LIN {X 0,Y 304.363,Z 602.903,A -85,B 0,C 180,E1 -16113.309,E2 -16113.309} C_VEL
LIN {X 0,Y 304.825,Z 598.921,A -85,B 0,C 180,E1 -16115.292,E2 -16115.292} C_VEL
LIN {X 0,Y 305.684,Z 593.946,A -85,B 0,C 180,E1 -16117.265,E2 -16117.265} C_VEL
LIN {X 0,Y 306.926,Z 586.616,A -85,B 0,C 180,E1 -16119.625,E2 -16119.625} C_VEL
LIN {X 0,Y 308.147,Z 578.097,A -85,B 0,C 180,E1 -16121.845,E2 -16121.845} C_VEL
LIN {X 0,Y 309.957,Z 568.895,A -85,B 0,C 180,E1 -16123.773,E2 -16123.773} C_VEL
LIN {X 0,Y 311.67,Z 558.74,A -85,B 0,C 180,E1 -16125.532,E2 -16125.532} C_VEL
LIN {X 0,Y 313.434,Z 547.553,A -85,B 0,C 180,E1 -16127.115,E2 -16127.115} C_VEL
LIN {X 0,Y 314.915,Z 536.756,A -85,B 0,C 180,E1 -16128.375,E2 -16128.375} C_VEL
LIN {X 0,Y 316.351,Z 525.204,A -85,B 0,C 180,E1 -16129.465,E2 -16129.465} C_VEL
LIN {X 0,Y 317.646,Z 512.743,A -85,B 0,C 180,E1 -16130.394,E2 -16130.394} C_VEL
LIN {X 0,Y 318.767,Z 498.862,A -85,B 0,C 180,E1 -16131.163,E2 -16131.163} C_VEL
LIN {X 0,Y 319.468,Z 485.64,A -85,B 0,C 180,E1 -16131.665,E2 -16131.665} C_VEL
LIN {X 0,Y 322.236,Z 387.309,A -85,B 0,C 180,E1 -16133.852,E2 -16133.852} C_VEL
LIN {X 0,Y 314.712,Z 368.239,A -85,B 0,C 180,E1 -16135.033,E2 -16135.033} C_VEL
LIN {X 0,Y 307.818,Z 353.094,A -85,B 0,C 180,E1 -16136.117,E2 -16136.117} C_VEL
LIN {X 0,Y 306.342,Z 349.731,A -85,B 0,C 180,E1 -16136.399,E2 -16136.399} C_VEL
LIN {X 0,Y 305.459,Z 346.064,A -85,B 0,C 180,E1 -16137.676,E2 -16137.676} C_VEL
LIN {X 0,Y 305.437,Z 346.065,A -85,B 0,C 180,E1 -16141.953,E2 -16141.953} C_VEL
LIN {X 0,Y 305.423,Z 346.063,A -85,B 0,C 180,E1 -16142.702,E2 -16142.702} C_VEL
LIN {X 0,Y 304.77,Z 346.147,A -85,B 0,C 180,E1 -16143.803,E2 -16143.803} C_VEL
LIN {X 0,Y 301.908,Z 346.503,A -85,B 0,C 180,E1 -16145.596,E2 -16145.596} C_VEL
LIN {X 0,Y 299.479,Z 346.804,A -85,B 0,C 180,E1 -16147.05,E2 -16147.05} C_VEL
LIN {X 0,Y 298.449,Z 346.935,A -85,B 0,C 180,E1 -16148.177,E2 -16148.177} C_VEL
LIN {X 0,Y 298.372,Z 346.94,A -85,B 0,C 180,E1 -16148.559,E2 -16148.559} C_VEL
LIN {X 0,Y 298.349,Z 346.944,A -85,B 0,C 180,E1 -16151.268,E2 -16151.268} C_VEL
LIN {X 0,Y 298.357,Z 346.94,A -85,B 0,C 180,E1 -16155.035,E2 -16155.035} C_VEL
LIN {X 0,Y 298.35,Z 346.941,A -85,B 0,C 180,E1 -16158.921,E2 -16158.921} C_VEL
LIN {X 0,Y 298.429,Z 346.93,A -85,B 0,C 180,E1 -16163.197,E2 -16163.197} C_VEL
LIN {X 0,Y 298.395,Z 346.929,A -85,B 0,C 180,E1 -16167.199,E2 -16167.199} C_VEL
LIN {X 0,Y 298.366,Z 346.942,A -85,B 0,C 180,E1 -16170.638,E2 -16170.638} C_VEL
LIN {X 0,Y 298.423,Z 346.937,A -85,B 0,C 180,E1 -16174.918,E2 -16174.918} C_VEL
LIN {X 0,Y 298.401,Z 346.924,A -85,B 0,C 180,E1 -16177.862,E2 -16177.862} C_VEL
LIN {X 0,Y 298.462,Z 346.907,A -85,B 0,C 180,E1 -16180.751,E2 -16180.751} C_VEL
LIN {X 0,Y 298.513,Z 346.923,A -85,B 0,C 180,E1 -16184.99,E2 -16184.99} C_VEL
LIN {X 0,Y 298.585,Z 346.881,A -85,B 0,C 180,E1 -16189.146,E2 -16189.146} C_VEL
LIN {X 0,Y 298.7,Z 346.893,A -85,B 0,C 180,E1 -16191.884,E2 -16191.884} C_VEL
LIN {X 0,Y 298.637,Z 346.908,A -85,B 0,C 180,E1 -16194.598,E2 -16194.598} C_VEL
LIN {X 0,Y 298.909,Z 346.876,A -85,B 0,C 180,E1 -16198.652,E2 -16198.652} C_VEL
LIN {X 0,Y 298.916,Z 346.867,A -85,B 0,C 180,E1 -16201.347,E2 -16201.347} C_VEL
LIN {X 0,Y 298.738,Z 346.896,A -85,B 0,C 180,E1 -16206.755,E2 -16206.755} C_VEL
LIN {X 0,Y 298.628,Z 346.909,A -85,B 0,C 180,E1 -16209.482,E2 -16209.482} C_VEL
LIN {X 0,Y 298.555,Z 346.918,A -85,B 0,C 180,E1 -16213.615,E2 -16213.615} C_VEL
LIN {X 0,Y 298.551,Z 346.921,A -85,B 0,C 180,E1 -16216.408,E2 -16216.408} C_VEL
LIN {X 0,Y 298.513,Z 346.925,A -85,B 0,C 180,E1 -16219.654,E2 -16219.654} C_VEL
LIN {X 0,Y 298.428,Z 346.937,A -85,B 0,C 180,E1 -16223.6,E2 -16223.6} C_VEL
LIN {X 0,Y 298.455,Z 346.933,A -85,B 0,C 180,E1 -16226.577,E2 -16226.577} C_VEL
LIN {X 0,Y 298.404,Z 346.938,A -85,B 0,C 180,E1 -16229.643,E2 -16229.643} C_VEL
LIN {X 0,Y 298.394,Z 346.939,A -85,B 0,C 180,E1 -16232.8,E2 -16232.8} C_VEL
LIN {X 0,Y 298.466,Z 346.934,A -85,B 0,C 180,E1 -16236.812,E2 -16236.812} C_VEL
LIN {X 0,Y 298.388,Z 346.944,A -85,B 0,C 180,E1 -16241.087,E2 -16241.087} C_VEL
LIN {X 0,Y 298.399,Z 346.943,A -85,B 0,C 180,E1 -16243.103,E2 -16243.103} C_VEL
LIN {X 0,Y 298.403,Z 346.94,A -85,B 0,C 180,E1 -16246.92,E2 -16246.92} C_VEL
LIN {X 0,Y 298.415,Z 346.943,A -85,B 0,C 180,E1 -16251.003,E2 -16251.003} C_VEL
LIN {X 0,Y 298.461,Z 347.007,A -85,B 0,C 180,E1 -16252.911,E2 -16252.911} C_VEL
LIN {X 0,Y 301.04,Z 357.568,A -85,B 0,C 180,E1 -16256.244,E2 -16256.244} C_VEL
LIN {X 0,Y 302.57,Z 364.284,A -85,B 0,C 180,E1 -16258.265,E2 -16258.265} C_VEL
LIN {X 0,Y 310.151,Z 382.609,A -85,B 0,C 180,E1 -16259.525,E2 -16259.525} C_VEL
LIN {X 0,Y 311.298,Z 386.467,A -85,B 0,C 180,E1 -16259.737,E2 -16259.737} C_VEL
LIN {X 0,Y 315.336,Z 412.615,A -85,B 0,C 180,E1 -16260.783,E2 -16260.783} C_VEL
LIN {X 0,Y 312.715,Z 502.779,A -85,B 0,C 180,E1 -16262.838,E2 -16262.838} C_VEL
LIN {X 0,Y 311.634,Z 517.379,A -85,B 0,C 180,E1 -16263.415,E2 -16263.415} C_VEL
LIN {X 0,Y 310.265,Z 531.359,A -85,B 0,C 180,E1 -16264.238,E2 -16264.238} C_VEL
LIN {X 0,Y 308.634,Z 544.36,A -85,B 0,C 180,E1 -16265.265,E2 -16265.265} C_VEL
LIN {X 0,Y 307.008,Z 556.448,A -85,B 0,C 180,E1 -16266.495,E2 -16266.495} C_VEL
LIN {X 0,Y 305.076,Z 568.504,A -85,B 0,C 180,E1 -16268.016,E2 -16268.016} C_VEL
LIN {X 0,Y 303.186,Z 579.067,A -85,B 0,C 180,E1 -16269.653,E2 -16269.653} C_VEL
LIN {X 0,Y 301.353,Z 589.573,A -85,B 0,C 180,E1 -16271.649,E2 -16271.649} C_VEL
LIN {X 0,Y 299.829,Z 598.233,A -85,B 0,C 180,E1 -16273.663,E2 -16273.663} C_VEL
LIN {X 0,Y 298.739,Z 605.428,A -85,B 0,C 180,E1 -16275.699,E2 -16275.699} C_VEL
LIN {X 0,Y 297.812,Z 611.401,A -85,B 0,C 180,E1 -16277.738,E2 -16277.738} C_VEL
LIN {X 0,Y 297.007,Z 617.772,A -85,B 0,C 180,E1 -16280.466,E2 -16280.466} C_VEL
LIN {X 0,Y 296.658,Z 622.48,A -85,B 0,C 180,E1 -16283.197,E2 -16283.197} C_VEL
LIN {X 0,Y 296.526,Z 625.665,A -85,B 0,C 180,E1 -16285.923,E2 -16285.923} C_VEL
LIN {X 0,Y 296.536,Z 626.733,A -85,B 0,C 180,E1 -16287.283,E2 -16287.283} C_VEL
LIN {X 0,Y 296.518,Z 627.85,A -85,B 0,C 180,E1 -16290,E2 -16290} C_VEL
LIN {X 0,Y 296.522,Z 627.627,A -85,B 0,C 180,E1 -16292.717,E2 -16292.717} C_VEL
LIN {X 0,Y 296.545,Z 626.01,A -85,B 0,C 180,E1 -16295.509,E2 -16295.509} C_VEL
LIN {X 0,Y 296.848,Z 623.148,A -85,B 0,C 180,E1 -16298.167,E2 -16298.167} C_VEL
LIN {X 0,Y 297.481,Z 618.79,A -85,B 0,C 180,E1 -16300.895,E2 -16300.895} C_VEL
LIN {X 0,Y 298.313,Z 614.495,A -85,B 0,C 180,E1 -16302.933,E2 -16302.933} C_VEL
LIN {X 0,Y 299.631,Z 608.255,A -85,B 0,C 180,E1 -16305.3,E2 -16305.3} C_VEL
LIN {X 0,Y 301.29,Z 600.498,A -85,B 0,C 180,E1 -16307.653,E2 -16307.653} C_VEL
LIN {X 0,Y 303.189,Z 592.422,A -85,B 0,C 180,E1 -16309.64,E2 -16309.64} C_VEL
LIN {X 0,Y 305.442,Z 582.706,A -85,B 0,C 180,E1 -16311.602,E2 -16311.602} C_VEL
LIN {X 0,Y 307.906,Z 571.94,A -85,B 0,C 180,E1 -16313.365,E2 -16313.365} C_VEL
LIN {X 0,Y 310.107,Z 561.08,A -85,B 0,C 180,E1 -16314.822,E2 -16314.822} C_VEL
LIN {X 0,Y 312.306,Z 548.346,A -85,B 0,C 180,E1 -16316.208,E2 -16316.208} C_VEL
LIN {X 0,Y 314.459,Z 534.587,A -85,B 0,C 180,E1 -16317.359,E2 -16317.359} C_VEL
LIN {X 0,Y 316.285,Z 520.471,A -85,B 0,C 180,E1 -16318.222,E2 -16318.222} C_VEL
LIN {X 0,Y 317.548,Z 506.55,A -85,B 0,C 180,E1 -16318.821,E2 -16318.821} C_VEL
LIN {X 0,Y 318.35,Z 489.027,A -85,B 0,C 180,E1 -16319.286,E2 -16319.286} C_VEL
LIN {X 0,Y 320.82,Z 413.586,A -85,B 0,C 180,E1 -16320.97,E2 -16320.97} C_VEL
LIN {X 0,Y 317.139,Z 393.638,A -85,B 0,C 180,E1 -16321.932,E2 -16321.932} C_VEL
LIN {X 0,Y 309.16,Z 376.1,A -85,B 0,C 180,E1 -16323.418,E2 -16323.418} C_VEL
LIN {X 0,Y 304.356,Z 366.77,A -85,B 0,C 180,E1 -16324.329,E2 -16324.329} C_VEL
LIN {X 0,Y 302.976,Z 363.672,A -85,B 0,C 180,E1 -16324.658,E2 -16324.658} C_VEL
LIN {X 0,Y 300.143,Z 352.926,A -85,B 0,C 180,E1 -16328.333,E2 -16328.333} C_VEL
LIN {X 0,Y 298.424,Z 346.939,A -85,B 0,C 180,E1 -16330.556,E2 -16330.556} C_VEL
LIN {X 0,Y 298.399,Z 346.937,A -85,B 0,C 180,E1 -16333.104,E2 -16333.104} C_VEL
LIN {X 0,Y 298.404,Z 346.939,A -85,B 0,C 180,E1 -16336.921,E2 -16336.921} C_VEL
LIN {X 0,Y 298.416,Z 346.932,A -85,B 0,C 180,E1 -16341.004,E2 -16341.004} C_VEL
LIN {X 0,Y 298.433,Z 346.929,A -85,B 0,C 180,E1 -16343.933,E2 -16343.933} C_VEL
LIN {X 0,Y 298.39,Z 346.94,A -85,B 0,C 180,E1 -16347.986,E2 -16347.986} C_VEL
LIN {X 0,Y 298.424,Z 346.937,A -85,B 0,C 180,E1 -16351.901,E2 -16351.901} C_VEL
LIN {X 0,Y 298.449,Z 346.932,A -85,B 0,C 180,E1 -16354.921,E2 -16354.921} C_VEL
LIN {X 0,Y 298.442,Z 346.932,A -85,B 0,C 180,E1 -16359.315,E2 -16359.315} C_VEL
LIN {X 0,Y 298.541,Z 346.913,A -85,B 0,C 180,E1 -16362.18,E2 -16362.18} C_VEL
LIN {X 0,Y 298.596,Z 346.914,A -85,B 0,C 180,E1 -16364.995,E2 -16364.995} C_VEL
LIN {X 0,Y 298.594,Z 346.915,A -85,B 0,C 180,E1 -16369.147,E2 -16369.147} C_VEL
LIN {X 0,Y 298.701,Z 346.891,A -85,B 0,C 180,E1 -16371.885,E2 -16371.885} C_VEL
LIN {X 0,Y 298.634,Z 346.91,A -85,B 0,C 180,E1 -16374.599,E2 -16374.599} C_VEL
LIN {X 0,Y 298.917,Z 346.875,A -85,B 0,C 180,E1 -16378.653,E2 -16378.653} C_VEL
LIN {X 0,Y 298.91,Z 346.866,A -85,B 0,C 180,E1 -16381.348,E2 -16381.348} C_VEL
LIN {X 0,Y 298.636,Z 346.907,A -85,B 0,C 180,E1 -16385.402,E2 -16385.402} C_VEL
LIN {X 0,Y 298.701,Z 346.897,A -85,B 0,C 180,E1 -16388.116,E2 -16388.116} C_VEL
LIN {X 0,Y 298.548,Z 346.912,A -85,B 0,C 180,E1 -16392.232,E2 -16392.232} C_VEL
LIN {X 0,Y 298.526,Z 346.922,A -85,B 0,C 180,E1 -16395.15,E2 -16395.15} C_VEL
LIN {X 0,Y 298.432,Z 346.932,A -85,B 0,C 180,E1 -16399.61,E2 -16399.61} C_VEL
LIN {X 0,Y 298.384,Z 346.94,A -85,B 0,C 180,E1 -16403.604,E2 -16403.604} C_VEL
LIN {X 0,Y 298.404,Z 346.939,A -85,B 0,C 180,E1 -16406.583,E2 -16406.583} C_VEL
LIN {X 0,Y 298.358,Z 346.915,A -85,B 0,C 180,E1 -16409.648,E2 -16409.648} C_VEL
LIN {X 0,Y 298.395,Z 346.937,A -85,B 0,C 180,E1 -16412.801,E2 -16412.801} C_VEL
LIN {X 0,Y 298.43,Z 346.912,A -85,B 0,C 180,E1 -16416.803,E2 -16416.803} C_VEL
LIN {X 0,Y 298.377,Z 346.943,A -85,B 0,C 180,E1 -16419.492,E2 -16419.492} C_VEL
LIN {X 0,Y 298.372,Z 346.942,A -85,B 0,C 180,E1 -16423.097,E2 -16423.097} C_VEL
LIN {X 0,Y 298.373,Z 346.938,A -85,B 0,C 180,E1 -16426.915,E2 -16426.915} C_VEL
LIN {X 0,Y 298.382,Z 347.116,A -85,B 0,C 180,E1 -16428.587,E2 -16428.587} C_VEL
LIN {X 0,Y 299.447,Z 350.821,A -85,B 0,C 180,E1 -16429.946,E2 -16429.946} C_VEL
LIN {X 0,Y 306.822,Z 364.05,A -85,B 0,C 180,E1 -16431.369,E2 -16431.369} C_VEL
LIN {X 0,Y 314.318,Z 378.638,A -85,B 0,C 180,E1 -16432.754,E2 -16432.754} C_VEL
LIN {X 0,Y 321.41,Z 394.73,A -85,B 0,C 180,E1 -16434.044,E2 -16434.044} C_VEL
LIN {X 0,Y 318.349,Z 486.508,A -85,B 0,C 180,E1 -16436.121,E2 -16436.121} C_VEL
LIN {X 0,Y 317.381,Z 500.566,A -85,B 0,C 180,E1 -16436.671,E2 -16436.671} C_VEL
LIN {X 0,Y 315.86,Z 514.254,A -85,B 0,C 180,E1 -16437.44,E2 -16437.44} C_VEL
LIN {X 0,Y 314.012,Z 527.678,A -85,B 0,C 180,E1 -16438.468,E2 -16438.468} C_VEL
LIN {X 0,Y 311.976,Z 540.359,A -85,B 0,C 180,E1 -16439.731,E2 -16439.731} C_VEL
LIN {X 0,Y 309.759,Z 551.972,A -85,B 0,C 180,E1 -16441.175,E2 -16441.175} C_VEL
LIN {X 0,Y 307.517,Z 562.596,A -85,B 0,C 180,E1 -16442.801,E2 -16442.801} C_VEL
LIN {X 0,Y 305.249,Z 573.118,A -85,B 0,C 180,E1 -16444.79,E2 -16444.79} C_VEL
LIN {X 0,Y 303.114,Z 581.766,A -85,B 0,C 180,E1 -16446.786,E2 -16446.786} C_VEL
LIN {X 0,Y 301.296,Z 589.273,A -85,B 0,C 180,E1 -16448.915,E2 -16448.915} C_VEL
LIN {X 0,Y 299.981,Z 594.86,A -85,B 0,C 180,E1 -16450.853,E2 -16450.853} C_VEL
LIN {X 0,Y 298.502,Z 601.166,A -85,B 0,C 180,E1 -16453.589,E2 -16453.589} C_VEL
LIN {X 0,Y 297.476,Z 605.807,A -85,B 0,C 180,E1 -16456.334,E2 -16456.334} C_VEL
LIN {X 0,Y 296.785,Z 608.93,A -85,B 0,C 180,E1 -16459.08,E2 -16459.08} C_VEL
LIN {X 0,Y 296.556,Z 610.669,A -85,B 0,C 180,E1 -16461.825,E2 -16461.825} C_VEL
LIN {X 0,Y 296.535,Z 611.079,A -85,B 0,C 180,E1 -16464.56,E2 -16464.56} C_VEL
LIN {X 0,Y 296.561,Z 610.178,A -85,B 0,C 180,E1 -16467.283,E2 -16467.283} C_VEL
LIN {X 0,Y 296.616,Z 607.957,A -85,B 0,C 180,E1 -16470,E2 -16470} C_VEL
LIN {X 0,Y 296.994,Z 604.356,A -85,B 0,C 180,E1 -16472.713,E2 -16472.713} C_VEL
LIN {X 0,Y 297.702,Z 600.672,A -85,B 0,C 180,E1 -16474.74,E2 -16474.74} C_VEL
LIN {X 0,Y 298.325,Z 596.116,A -85,B 0,C 180,E1 -16476.765,E2 -16476.765} C_VEL
LIN {X 0,Y 299.539,Z 589.482,A -85,B 0,C 180,E1 -16479.113,E2 -16479.113} C_VEL
LIN {X 0,Y 300.645,Z 582.541,A -85,B 0,C 180,E1 -16481.119,E2 -16481.119} C_VEL
LIN {X 0,Y 301.843,Z 575.685,A -85,B 0,C 180,E1 -16482.779,E2 -16482.779} C_VEL
LIN {X 0,Y 303.733,Z 565.943,A -85,B 0,C 180,E1 -16484.746,E2 -16484.746} C_VEL
LIN {X 0,Y 305.554,Z 555.143,A -85,B 0,C 180,E1 -16486.537,E2 -16486.537} C_VEL
LIN {X 0,Y 307.16,Z 544.449,A -85,B 0,C 180,E1 -16487.992,E2 -16487.992} C_VEL
LIN {X 0,Y 309.053,Z 531.337,A -85,B 0,C 180,E1 -16489.425,E2 -16489.425} C_VEL
LIN {X 0,Y 310.579,Z 518.341,A -85,B 0,C 180,E1 -16490.533,E2 -16490.533} C_VEL
LIN {X 0,Y 311.912,Z 504.14,A -85,B 0,C 180,E1 -16491.435,E2 -16491.435} C_VEL
LIN {X 0,Y 312.834,Z 490.019,A -85,B 0,C 180,E1 -16492.061,E2 -16492.061} C_VEL
LIN {X 0,Y 313.514,Z 471.195,A -85,B 0,C 180,E1 -16492.556,E2 -16492.556} C_VEL
LIN {X 0,Y 315.783,Z 388.813,A -85,B 0,C 180,E1 -16494.411,E2 -16494.411} C_VEL
LIN {X 0,Y 308.537,Z 370.431,A -85,B 0,C 180,E1 -16495.59,E2 -16495.59} C_VEL
LIN {X 0,Y 300.495,Z 353.052,A -85,B 0,C 180,E1 -16496.9,E2 -16496.9} C_VEL
LIN {X 0,Y 299.148,Z 350.04,A -85,B 0,C 180,E1 -16497.148,E2 -16497.148} C_VEL
LIN {X 0,Y 298.473,Z 346.934,A -85,B 0,C 180,E1 -16498.286,E2 -16498.286} C_VEL
LIN {X 0,Y 298.395,Z 346.94,A -85,B 0,C 180,E1 -16502.8,E2 -16502.8} C_VEL
LIN {X 0,Y 298.406,Z 346.94,A -85,B 0,C 180,E1 -16506.072,E2 -16506.072} C_VEL
LIN {X 0,Y 298.372,Z 346.94,A -85,B 0,C 180,E1 -16508.559,E2 -16508.559} C_VEL
LIN {X 0,Y 297.724,Z 347.022,A -85,B 0,C 180,E1 -16509.686,E2 -16509.686} C_VEL
LIN {X 0,Y 294.877,Z 347.382,A -85,B 0,C 180,E1 -16511.521,E2 -16511.521} C_VEL
LIN {X 0,Y 292.438,Z 347.685,A -85,B 0,C 180,E1 -16513.01,E2 -16513.01} C_VEL
LIN {X 0,Y 291.373,Z 347.815,A -85,B 0,C 180,E1 -16514.163,E2 -16514.163} C_VEL
LIN {X 0,Y 291.277,Z 347.824,A -85,B 0,C 180,E1 -16514.554,E2 -16514.554} C_VEL
LIN {X 0,Y 291.297,Z 347.819,A -85,B 0,C 180,E1 -16518.411,E2 -16518.411} C_VEL
LIN {X 0,Y 291.311,Z 347.821,A -85,B 0,C 180,E1 -16521.151,E2 -16521.151} C_VEL
LIN {X 0,Y 291.358,Z 347.819,A -85,B 0,C 180,E1 -16524.625,E2 -16524.625} C_VEL
LIN {X 0,Y 291.368,Z 347.806,A -85,B 0,C 180,E1 -16527.95,E2 -16527.95} C_VEL
LIN {X 0,Y 291.317,Z 347.817,A -85,B 0,C 180,E1 -16531.151,E2 -16531.151} C_VEL
LIN {X 0,Y 291.348,Z 347.815,A -85,B 0,C 180,E1 -16534.265,E2 -16534.265} C_VEL
LIN {X 0,Y 291.36,Z 347.809,A -85,B 0,C 180,E1 -16537.297,E2 -16537.297} C_VEL
LIN {X 0,Y 291.391,Z 347.782,A -85,B 0,C 180,E1 -16540.265,E2 -16540.265} C_VEL
LIN {X 0,Y 291.476,Z 347.801,A -85,B 0,C 180,E1 -16544.682,E2 -16544.682} C_VEL
LIN {X 0,Y 291.53,Z 347.759,A -85,B 0,C 180,E1 -16548.88,E2 -16548.88} C_VEL
LIN {X 0,Y 291.654,Z 347.769,A -85,B 0,C 180,E1 -16551.686,E2 -16551.686} C_VEL
LIN {X 0,Y 291.606,Z 347.785,A -85,B 0,C 180,E1 -16554.467,E2 -16554.467} C_VEL
LIN {X 0,Y 291.877,Z 347.752,A -85,B 0,C 180,E1 -16558.62,E2 -16558.62} C_VEL
LIN {X 0,Y 291.882,Z 347.743,A -85,B 0,C 180,E1 -16561.379,E2 -16561.379} C_VEL
LIN {X 0,Y 291.69,Z 347.773,A -85,B 0,C 180,E1 -16566.919,E2 -16566.919} C_VEL
LIN {X 0,Y 291.57,Z 347.786,A -85,B 0,C 180,E1 -16569.713,E2 -16569.713} C_VEL
LIN {X 0,Y 291.525,Z 347.792,A -85,B 0,C 180,E1 -16573.95,E2 -16573.95} C_VEL
LIN {X 0,Y 291.489,Z 347.799,A -85,B 0,C 180,E1 -16576.817,E2 -16576.817} C_VEL
LIN {X 0,Y 291.452,Z 347.807,A -85,B 0,C 180,E1 -16579.874,E2 -16579.874} C_VEL
LIN {X 0,Y 291.375,Z 347.816,A -85,B 0,C 180,E1 -16584.207,E2 -16584.207} C_VEL
LIN {X 0,Y 291.399,Z 347.813,A -85,B 0,C 180,E1 -16587.274,E2 -16587.274} C_VEL
LIN {X 0,Y 291.325,Z 347.824,A -85,B 0,C 180,E1 -16590.438,E2 -16590.438} C_VEL
LIN {X 0,Y 291.345,Z 347.822,A -85,B 0,C 180,E1 -16593.698,E2 -16593.698} C_VEL
LIN {X 0,Y 291.396,Z 347.817,A -85,B 0,C 180,E1 -16597.259,E2 -16597.259} C_VEL
LIN {X 0,Y 291.335,Z 347.822,A -85,B 0,C 180,E1 -16600.642,E2 -16600.642} C_VEL
LIN {X 0,Y 291.29,Z 347.827,A -85,B 0,C 180,E1 -16604.402,E2 -16604.402} C_VEL
LIN {X 0,Y 291.327,Z 347.82,A -85,B 0,C 180,E1 -16608.404,E2 -16608.404} C_VEL
LIN {X 0,Y 291.41,Z 347.925,A -85,B 0,C 180,E1 -16612.283,E2 -16612.283} C_VEL
LIN {X 0,Y 294.108,Z 358.827,A -85,B 0,C 180,E1 -16615.837,E2 -16615.837} C_VEL
LIN {X 0,Y 295.375,Z 364.297,A -85,B 0,C 180,E1 -16617.476,E2 -16617.476} C_VEL
LIN {X 0,Y 303.014,Z 382.178,A -85,B 0,C 180,E1 -16618.789,E2 -16618.789} C_VEL
LIN {X 0,Y 305.188,Z 388.485,A -85,B 0,C 180,E1 -16619.18,E2 -16619.18} C_VEL
LIN {X 0,Y 308.986,Z 413.438,A -85,B 0,C 180,E1 -16620.204,E2 -16620.204} C_VEL
LIN {X 0,Y 306.319,Z 502.381,A -85,B 0,C 180,E1 -16622.269,E2 -16622.269} C_VEL
LIN {X 0,Y 305.207,Z 517.046,A -85,B 0,C 180,E1 -16622.856,E2 -16622.856} C_VEL
LIN {X 0,Y 303.732,Z 531.63,A -85,B 0,C 180,E1 -16623.734,E2 -16623.734} C_VEL
LIN {X 0,Y 301.93,Z 545.418,A -85,B 0,C 180,E1 -16624.862,E2 -16624.862} C_VEL
LIN {X 0,Y 300.182,Z 557.645,A -85,B 0,C 180,E1 -16626.159,E2 -16626.159} C_VEL
LIN {X 0,Y 298.254,Z 569.141,A -85,B 0,C 180,E1 -16627.668,E2 -16627.668} C_VEL
LIN {X 0,Y 296.119,Z 580.517,A -85,B 0,C 180,E1 -16629.508,E2 -16629.508} C_VEL
LIN {X 0,Y 294.259,Z 590.684,A -85,B 0,C 180,E1 -16631.551,E2 -16631.551} C_VEL
LIN {X 0,Y 292.762,Z 599.004,A -85,B 0,C 180,E1 -16633.582,E2 -16633.582} C_VEL
LIN {X 0,Y 291.607,Z 606.165,A -85,B 0,C 180,E1 -16635.698,E2 -16635.698} C_VEL
LIN {X 0,Y 290.547,Z 612.851,A -85,B 0,C 180,E1 -16638.135,E2 -16638.135} C_VEL
LIN {X 0,Y 289.824,Z 618.782,A -85,B 0,C 180,E1 -16640.931,E2 -16640.931} C_VEL
LIN {X 0,Y 289.581,Z 622.209,A -85,B 0,C 180,E1 -16643.03,E2 -16643.03} C_VEL
LIN {X 0,Y 289.428,Z 625.423,A -85,B 0,C 180,E1 -16645.822,E2 -16645.822} C_VEL
LIN {X 0,Y 289.417,Z 627.241,A -85,B 0,C 180,E1 -16648.609,E2 -16648.609} C_VEL
LIN {X 0,Y 289.412,Z 627.709,A -85,B 0,C 180,E1 -16651.392,E2 -16651.392} C_VEL
LIN {X 0,Y 289.391,Z 626.841,A -85,B 0,C 180,E1 -16654.178,E2 -16654.178} C_VEL
LIN {X 0,Y 289.573,Z 624.632,A -85,B 0,C 180,E1 -16656.97,E2 -16656.97} C_VEL
LIN {X 0,Y 290.053,Z 621.03,A -85,B 0,C 180,E1 -16659.765,E2 -16659.765} C_VEL
LIN {X 0,Y 290.976,Z 615.936,A -85,B 0,C 180,E1 -16662.555,E2 -16662.555} C_VEL
LIN {X 0,Y 292.129,Z 611.025,A -85,B 0,C 180,E1 -16664.632,E2 -16664.632} C_VEL
LIN {X 0,Y 293.668,Z 603.983,A -85,B 0,C 180,E1 -16667.048,E2 -16667.048} C_VEL
LIN {X 0,Y 295.799,Z 595.283,A -85,B 0,C 180,E1 -16669.429,E2 -16669.429} C_VEL
LIN {X 0,Y 298.064,Z 586.203,A -85,B 0,C 180,E1 -16671.437,E2 -16671.437} C_VEL
LIN {X 0,Y 300.703,Z 575.226,A -85,B 0,C 180,E1 -16673.411,E2 -16673.411} C_VEL
LIN {X 0,Y 303.177,Z 563.949,A -85,B 0,C 180,E1 -16675.045,E2 -16675.045} C_VEL
LIN {X 0,Y 305.453,Z 551.759,A -85,B 0,C 180,E1 -16676.474,E2 -16676.474} C_VEL
LIN {X 0,Y 307.444,Z 539.939,A -85,B 0,C 180,E1 -16677.575,E2 -16677.575} C_VEL
LIN {X 0,Y 309.341,Z 527.055,A -85,B 0,C 180,E1 -16678.497,E2 -16678.497} C_VEL
LIN {X 0,Y 310.985,Z 512.379,A -85,B 0,C 180,E1 -16679.256,E2 -16679.256} C_VEL
LIN {X 0,Y 311.97,Z 497.873,A -85,B 0,C 180,E1 -16679.75,E2 -16679.75} C_VEL
LIN {X 0,Y 314.892,Z 415.193,A -85,B 0,C 180,E1 -16681.627,E2 -16681.627} C_VEL
LIN {X 0,Y 311.485,Z 396.413,A -85,B 0,C 180,E1 -16682.556,E2 -16682.556} C_VEL
LIN {X 0,Y 304.109,Z 380.105,A -85,B 0,C 180,E1 -16683.981,E2 -16683.981} C_VEL
LIN {X 0,Y 297.473,Z 367.151,A -85,B 0,C 180,E1 -16685.297,E2 -16685.297} C_VEL
LIN {X 0,Y 295.704,Z 363.436,A -85,B 0,C 180,E1 -16685.718,E2 -16685.718} C_VEL
LIN {X 0,Y 292.928,Z 353.359,A -85,B 0,C 180,E1 -16689.325,E2 -16689.325} C_VEL
LIN {X 0,Y 291.337,Z 347.818,A -85,B 0,C 180,E1 -16691.499,E2 -16691.499} C_VEL
LIN {X 0,Y 291.29,Z 347.821,A -85,B 0,C 180,E1 -16695.598,E2 -16695.598} C_VEL
LIN {X 0,Y 291.335,Z 347.819,A -85,B 0,C 180,E1 -16699.358,E2 -16699.358} C_VEL
LIN {X 0,Y 291.426,Z 347.805,A -85,B 0,C 180,E1 -16702.923,E2 -16702.923} C_VEL
LIN {X 0,Y 291.345,Z 347.814,A -85,B 0,C 180,E1 -16706.302,E2 -16706.302} C_VEL
LIN {X 0,Y 291.37,Z 347.809,A -85,B 0,C 180,E1 -16710.267,E2 -16710.267} C_VEL
LIN {X 0,Y 291.376,Z 347.808,A -85,B 0,C 180,E1 -16714.268,E2 -16714.268} C_VEL
LIN {X 0,Y 291.375,Z 347.808,A -85,B 0,C 180,E1 -16717.299,E2 -16717.299} C_VEL
LIN {X 0,Y 291.46,Z 347.805,A -85,B 0,C 180,E1 -16720.271,E2 -16720.271} C_VEL
LIN {X 0,Y 291.558,Z 347.792,A -85,B 0,C 180,E1 -16724.624,E2 -16724.624} C_VEL
LIN {X 0,Y 291.538,Z 347.794,A -85,B 0,C 180,E1 -16728.881,E2 -16728.881} C_VEL
LIN {X 0,Y 291.654,Z 347.769,A -85,B 0,C 180,E1 -16731.687,E2 -16731.687} C_VEL
LIN {X 0,Y 291.603,Z 347.786,A -85,B 0,C 180,E1 -16734.468,E2 -16734.468} C_VEL
LIN {X 0,Y 291.883,Z 347.751,A -85,B 0,C 180,E1 -16738.621,E2 -16738.621} C_VEL
LIN {X 0,Y 291.878,Z 347.741,A -85,B 0,C 180,E1 -16741.38,E2 -16741.38} C_VEL
LIN {X 0,Y 291.65,Z 347.767,A -85,B 0,C 180,E1 -16746.537,E2 -16746.537} C_VEL
LIN {X 0,Y 291.572,Z 347.791,A -85,B 0,C 180,E1 -16749.714,E2 -16749.714} C_VEL
LIN {X 0,Y 291.485,Z 347.803,A -85,B 0,C 180,E1 -16753.953,E2 -16753.953} C_VEL
LIN {X 0,Y 291.404,Z 347.801,A -85,B 0,C 180,E1 -16756.823,E2 -16756.823} C_VEL
LIN {X 0,Y 291.394,Z 347.806,A -85,B 0,C 180,E1 -16759.842,E2 -16759.842} C_VEL
LIN {X 0,Y 291.329,Z 347.814,A -85,B 0,C 180,E1 -16764.212,E2 -16764.212} C_VEL
LIN {X 0,Y 291.331,Z 347.82,A -85,B 0,C 180,E1 -16767.281,E2 -16767.281} C_VEL
LIN {X 0,Y 291.303,Z 347.79,A -85,B 0,C 180,E1 -16770.441,E2 -16770.441} C_VEL
LIN {X 0,Y 291.346,Z 347.82,A -85,B 0,C 180,E1 -16773.699,E2 -16773.699} C_VEL
LIN {X 0,Y 291.361,Z 347.794,A -85,B 0,C 180,E1 -16777.249,E2 -16777.249} C_VEL
LIN {X 0,Y 291.303,Z 347.82,A -85,B 0,C 180,E1 -16780.648,E2 -16780.648} C_VEL
LIN {X 0,Y 291.285,Z 347.825,A -85,B 0,C 180,E1 -16784.404,E2 -16784.404} C_VEL
LIN {X 0,Y 291.354,Z 347.911,A -85,B 0,C 180,E1 -16787.671,E2 -16787.671} C_VEL
LIN {X 0,Y 292.077,Z 350.81,A -85,B 0,C 180,E1 -16788.83,E2 -16788.83} C_VEL
LIN {X 0,Y 301.5,Z 367.369,A -85,B 0,C 180,E1 -16790.727,E2 -16790.727} C_VEL
LIN {X 0,Y 309.374,Z 382.932,A -85,B 0,C 180,E1 -16792.239,E2 -16792.239} C_VEL
LIN {X 0,Y 315.479,Z 396.981,A -85,B 0,C 180,E1 -16793.394,E2 -16793.394} C_VEL
LIN {X 0,Y 312.276,Z 487.181,A -85,B 0,C 180,E1 -16795.468,E2 -16795.468} C_VEL
LIN {X 0,Y 311.156,Z 501.833,A -85,B 0,C 180,E1 -16796.06,E2 -16796.06} C_VEL
LIN {X 0,Y 309.552,Z 515.82,A -85,B 0,C 180,E1 -16796.885,E2 -16796.885} C_VEL
LIN {X 0,Y 307.925,Z 527.152,A -85,B 0,C 180,E1 -16797.769,E2 -16797.769} C_VEL
LIN {X 0,Y 305.808,Z 539.981,A -85,B 0,C 180,E1 -16799.055,E2 -16799.055} C_VEL
LIN {X 0,Y 303.445,Z 551.693,A -85,B 0,C 180,E1 -16800.517,E2 -16800.517} C_VEL
LIN {X 0,Y 301.116,Z 562.398,A -85,B 0,C 180,E1 -16802.173,E2 -16802.173} C_VEL
LIN {X 0,Y 298.739,Z 572.987,A -85,B 0,C 180,E1 -16804.2,E2 -16804.2} C_VEL
LIN {X 0,Y 296.495,Z 581.691,A -85,B 0,C 180,E1 -16806.236,E2 -16806.236} C_VEL
LIN {X 0,Y 294.418,Z 589.822,A -85,B 0,C 180,E1 -16808.587,E2 -16808.587} C_VEL
LIN {X 0,Y 292.716,Z 596.655,A -85,B 0,C 180,E1 -16811.087,E2 -16811.087} C_VEL
LIN {X 0,Y 291.28,Z 602.527,A -85,B 0,C 180,E1 -16813.89,E2 -16813.89} C_VEL
LIN {X 0,Y 290.506,Z 605.913,A -85,B 0,C 180,E1 -16816,E2 -16816} C_VEL
LIN {X 0,Y 289.737,Z 609.075,A -85,B 0,C 180,E1 -16818.811,E2 -16818.811} C_VEL
LIN {X 0,Y 289.48,Z 610.847,A -85,B 0,C 180,E1 -16821.624,E2 -16821.624} C_VEL
LIN {X 0,Y 289.462,Z 611.289,A -85,B 0,C 180,E1 -16824.427,E2 -16824.427} C_VEL
LIN {X 0,Y 289.485,Z 610.419,A -85,B 0,C 180,E1 -16827.217,E2 -16827.217} C_VEL
LIN {X 0,Y 289.529,Z 608.232,A -85,B 0,C 180,E1 -16830,E2 -16830} C_VEL
LIN {X 0,Y 289.914,Z 604.665,A -85,B 0,C 180,E1 -16832.779,E2 -16832.779} C_VEL
LIN {X 0,Y 290.629,Z 601.019,A -85,B 0,C 180,E1 -16834.855,E2 -16834.855} C_VEL
LIN {X 0,Y 291.302,Z 596.485,A -85,B 0,C 180,E1 -16836.929,E2 -16836.929} C_VEL
LIN {X 0,Y 292.559,Z 589.898,A -85,B 0,C 180,E1 -16839.332,E2 -16839.332} C_VEL
LIN {X 0,Y 293.874,Z 581.728,A -85,B 0,C 180,E1 -16841.729,E2 -16841.729} C_VEL
LIN {X 0,Y 295.624,Z 573.187,A -85,B 0,C 180,E1 -16843.753,E2 -16843.753} C_VEL
LIN {X 0,Y 297.585,Z 562.846,A -85,B 0,C 180,E1 -16845.759,E2 -16845.759} C_VEL
LIN {X 0,Y 299.516,Z 551.296,A -85,B 0,C 180,E1 -16847.584,E2 -16847.584} C_VEL
LIN {X 0,Y 301.329,Z 539.739,A -85,B 0,C 180,E1 -16849.058,E2 -16849.058} C_VEL
LIN {X 0,Y 303.116,Z 527.029,A -85,B 0,C 180,E1 -16850.352,E2 -16850.352} C_VEL
LIN {X 0,Y 304.594,Z 513.848,A -85,B 0,C 180,E1 -16851.398,E2 -16851.398} C_VEL
LIN {X 0,Y 305.824,Z 500.269,A -85,B 0,C 180,E1 -16852.194,E2 -16852.194} C_VEL
LIN {X 0,Y 306.627,Z 486.374,A -85,B 0,C 180,E1 -16852.754,E2 -16852.754} C_VEL
LIN {X 0,Y 309.55,Z 390.783,A -85,B 0,C 180,E1 -16854.962,E2 -16854.962} C_VEL
LIN {X 0,Y 302.53,Z 372.918,A -85,B 0,C 180,E1 -16856.147,E2 -16856.147} C_VEL
LIN {X 0,Y 293.451,Z 353.513,A -85,B 0,C 180,E1 -16857.682,E2 -16857.682} C_VEL
LIN {X 0,Y 291.98,Z 350.319,A -85,B 0,C 180,E1 -16857.944,E2 -16857.944} C_VEL
LIN {X 0,Y 291.379,Z 347.817,A -85,B 0,C 180,E1 -16858.842,E2 -16858.842} C_VEL
LIN {X 0,Y 291.34,Z 347.819,A -85,B 0,C 180,E1 -16862.401,E2 -16862.401} C_VEL
LIN {X 0,Y 291.357,Z 347.818,A -85,B 0,C 180,E1 -16865.375,E2 -16865.375} C_VEL
LIN {X 0,Y 291.335,Z 347.818,A -85,B 0,C 180,E1 -16868.845,E2 -16868.845} C_VEL
LIN {X 0,Y 291.289,Z 347.823,A -85,B 0,C 180,E1 -16872.498,E2 -16872.498} C_VEL
LIN {X 0,Y 291.277,Z 347.824,A -85,B 0,C 180,E1 -16874.554,E2 -16874.554} C_VEL
LIN {X 0,Y 290.592,Z 347.909,A -85,B 0,C 180,E1 -16875.708,E2 -16875.708} C_VEL
LIN {X 0,Y 287.76,Z 348.263,A -85,B 0,C 180,E1 -16877.588,E2 -16877.588} C_VEL
LIN {X 0,Y 285.369,Z 348.561,A -85,B 0,C 180,E1 -16879.113,E2 -16879.113} C_VEL
LIN {X 0,Y 284.34,Z 348.691,A -85,B 0,C 180,E1 -16880.295,E2 -16880.295} C_VEL
LIN {X 0,Y 284.253,Z 348.696,A -85,B 0,C 180,E1 -16880.695,E2 -16880.695} C_VEL
LIN {X 0,Y 284.339,Z 348.693,A -85,B 0,C 180,E1 -16884.653,E2 -16884.653} C_VEL
LIN {X 0,Y 284.281,Z 348.695,A -85,B 0,C 180,E1 -16888.723,E2 -16888.723} C_VEL
LIN {X 0,Y 284.262,Z 348.691,A -85,B 0,C 180,E1 -16891.981,E2 -16891.981} C_VEL
LIN {X 0,Y 284.313,Z 348.695,A -85,B 0,C 180,E1 -16896.152,E2 -16896.152} C_VEL
LIN {X 0,Y 284.336,Z 348.659,A -85,B 0,C 180,E1 -16899.928,E2 -16899.928} C_VEL
LIN {X 0,Y 284.417,Z 348.682,A -85,B 0,C 180,E1 -16904.516,E2 -16904.516} C_VEL
LIN {X 0,Y 284.467,Z 348.639,A -85,B 0,C 180,E1 -16908.6,E2 -16908.6} C_VEL
LIN {X 0,Y 284.611,Z 348.645,A -85,B 0,C 180,E1 -16911.479,E2 -16911.479} C_VEL
LIN {X 0,Y 284.575,Z 348.662,A -85,B 0,C 180,E1 -16914.33,E2 -16914.33} C_VEL
LIN {X 0,Y 284.844,Z 348.628,A -85,B 0,C 180,E1 -16918.586,E2 -16918.586} C_VEL
LIN {X 0,Y 284.848,Z 348.619,A -85,B 0,C 180,E1 -16921.413,E2 -16921.413} C_VEL
LIN {X 0,Y 284.645,Z 348.651,A -85,B 0,C 180,E1 -16927.091,E2 -16927.091} C_VEL
LIN {X 0,Y 284.516,Z 348.664,A -85,B 0,C 180,E1 -16929.957,E2 -16929.957} C_VEL
LIN {X 0,Y 284.484,Z 348.668,A -85,B 0,C 180,E1 -16934.302,E2 -16934.302} C_VEL
LIN {X 0,Y 284.428,Z 348.68,A -85,B 0,C 180,E1 -16937.248,E2 -16937.248} C_VEL
LIN {X 0,Y 284.38,Z 348.687,A -85,B 0,C 180,E1 -16940.242,E2 -16940.242} C_VEL
LIN {X 0,Y 284.324,Z 348.692,A -85,B 0,C 180,E1 -16944.848,E2 -16944.848} C_VEL
LIN {X 0,Y 284.31,Z 348.696,A -85,B 0,C 180,E1 -16948.013,E2 -16948.013} C_VEL
LIN {X 0,Y 284.288,Z 348.702,A -85,B 0,C 180,E1 -16951.275,E2 -16951.275} C_VEL
LIN {X 0,Y 284.363,Z 348.689,A -85,B 0,C 180,E1 -16955.354,E2 -16955.354} C_VEL
LIN {X 0,Y 284.325,Z 348.692,A -85,B 0,C 180,E1 -16958.167,E2 -16958.167} C_VEL
LIN {X 0,Y 284.27,Z 348.703,A -85,B 0,C 180,E1 -16962.124,E2 -16962.124} C_VEL
LIN {X 0,Y 284.255,Z 348.702,A -85,B 0,C 180,E1 -16966.189,E2 -16966.189} C_VEL
LIN {X 0,Y 284.307,Z 348.696,A -85,B 0,C 180,E1 -16970.023,E2 -16970.023} C_VEL
LIN {X 0,Y 284.336,Z 348.82,A -85,B 0,C 180,E1 -16971.609,E2 -16971.609} C_VEL
LIN {X 0,Y 287.149,Z 359.786,A -85,B 0,C 180,E1 -16975.316,E2 -16975.316} C_VEL
LIN {X 0,Y 288.089,Z 363.978,A -85,B 0,C 180,E1 -16976.62,E2 -16976.62} C_VEL
LIN {X 0,Y 296.345,Z 382.976,A -85,B 0,C 180,E1 -16978.096,E2 -16978.096} C_VEL
LIN {X 0,Y 299.169,Z 390.791,A -85,B 0,C 180,E1 -16978.614,E2 -16978.614} C_VEL
LIN {X 0,Y 302.681,Z 414.399,A -85,B 0,C 180,E1 -16979.607,E2 -16979.607} C_VEL
LIN {X 0,Y 299.96,Z 501.961,A -85,B 0,C 180,E1 -16981.676,E2 -16981.676} C_VEL
LIN {X 0,Y 298.937,Z 515.949,A -85,B 0,C 180,E1 -16982.238,E2 -16982.238} C_VEL
LIN {X 0,Y 297.51,Z 529.625,A -85,B 0,C 180,E1 -16983.047,E2 -16983.047} C_VEL
LIN {X 0,Y 295.719,Z 542.913,A -85,B 0,C 180,E1 -16984.107,E2 -16984.107} C_VEL
LIN {X 0,Y 293.916,Z 555.233,A -85,B 0,C 180,E1 -16985.385,E2 -16985.385} C_VEL
LIN {X 0,Y 291.885,Z 567.41,A -85,B 0,C 180,E1 -16986.967,E2 -16986.967} C_VEL
LIN {X 0,Y 289.81,Z 578.088,A -85,B 0,C 180,E1 -16988.669,E2 -16988.669} C_VEL
LIN {X 0,Y 287.764,Z 588.687,A -85,B 0,C 180,E1 -16990.749,E2 -16990.749} C_VEL
LIN {X 0,Y 286.052,Z 597.426,A -85,B 0,C 180,E1 -16992.853,E2 -16992.853} C_VEL
LIN {X 0,Y 284.935,Z 604.698,A -85,B 0,C 180,E1 -16994.99,E2 -16994.99} C_VEL
LIN {X 0,Y 283.855,Z 610.731,A -85,B 0,C 180,E1 -16997.125,E2 -16997.125} C_VEL
LIN {X 0,Y 282.915,Z 617.16,A -85,B 0,C 180,E1 -16999.986,E2 -16999.986} C_VEL
LIN {X 0,Y 282.502,Z 621.934,A -85,B 0,C 180,E1 -17002.855,E2 -17002.855} C_VEL
LIN {X 0,Y 282.336,Z 625.18,A -85,B 0,C 180,E1 -17005.717,E2 -17005.717} C_VEL
LIN {X 0,Y 282.34,Z 627.022,A -85,B 0,C 180,E1 -17008.574,E2 -17008.574} C_VEL
LIN {X 0,Y 282.335,Z 627.514,A -85,B 0,C 180,E1 -17011.426,E2 -17011.426} C_VEL
LIN {X 0,Y 282.3,Z 626.668,A -85,B 0,C 180,E1 -17014.283,E2 -17014.283} C_VEL
LIN {X 0,Y 282.494,Z 624.482,A -85,B 0,C 180,E1 -17017.146,E2 -17017.146} C_VEL
LIN {X 0,Y 283.034,Z 620.905,A -85,B 0,C 180,E1 -17020.01,E2 -17020.01} C_VEL
LIN {X 0,Y 284.03,Z 615.838,A -85,B 0,C 180,E1 -17022.867,E2 -17022.867} C_VEL
LIN {X 0,Y 285.197,Z 610.955,A -85,B 0,C 180,E1 -17024.996,E2 -17024.996} C_VEL
LIN {X 0,Y 286.858,Z 603.943,A -85,B 0,C 180,E1 -17027.465,E2 -17027.465} C_VEL
LIN {X 0,Y 289.097,Z 595.28,A -85,B 0,C 180,E1 -17029.898,E2 -17029.898} C_VEL
LIN {X 0,Y 291.421,Z 586.241,A -85,B 0,C 180,E1 -17031.951,E2 -17031.951} C_VEL
LIN {X 0,Y 294.185,Z 575.314,A -85,B 0,C 180,E1 -17033.962,E2 -17033.962} C_VEL
LIN {X 0,Y 296.852,Z 563.671,A -85,B 0,C 180,E1 -17035.684,E2 -17035.684} C_VEL
LIN {X 0,Y 299.111,Z 552.028,A -85,B 0,C 180,E1 -17037.081,E2 -17037.081} C_VEL
LIN {X 0,Y 301.195,Z 540.318,A -85,B 0,C 180,E1 -17038.197,E2 -17038.197} C_VEL
LIN {X 0,Y 303.136,Z 527.619,A -85,B 0,C 180,E1 -17039.135,E2 -17039.135} C_VEL
LIN {X 0,Y 304.849,Z 513.261,A -85,B 0,C 180,E1 -17039.904,E2 -17039.904} C_VEL
LIN {X 0,Y 305.882,Z 499.431,A -85,B 0,C 180,E1 -17040.405,E2 -17040.405} C_VEL
LIN {X 0,Y 308.88,Z 415.528,A -85,B 0,C 180,E1 -17042.36,E2 -17042.36} C_VEL
LIN {X 0,Y 305.881,Z 399.169,A -85,B 0,C 180,E1 -17043.203,E2 -17043.203} C_VEL
LIN {X 0,Y 298.713,Z 383.369,A -85,B 0,C 180,E1 -17044.639,E2 -17044.639} C_VEL
LIN {X 0,Y 292.245,Z 370.667,A -85,B 0,C 180,E1 -17045.974,E2 -17045.974} C_VEL
LIN {X 0,Y 288.437,Z 363.28,A -85,B 0,C 180,E1 -17046.814,E2 -17046.814} C_VEL
LIN {X 0,Y 285.83,Z 353.86,A -85,B 0,C 180,E1 -17050.339,E2 -17050.339} C_VEL
LIN {X 0,Y 284.297,Z 348.699,A -85,B 0,C 180,E1 -17052.45,E2 -17052.45} C_VEL
LIN {X 0,Y 284.256,Z 348.698,A -85,B 0,C 180,E1 -17056.19,E2 -17056.19} C_VEL
LIN {X 0,Y 284.308,Z 348.692,A -85,B 0,C 180,E1 -17060.024,E2 -17060.024} C_VEL
LIN {X 0,Y 284.352,Z 348.683,A -85,B 0,C 180,E1 -17063.617,E2 -17063.617} C_VEL
LIN {X 0,Y 284.307,Z 348.69,A -85,B 0,C 180,E1 -17067.191,E2 -17067.191} C_VEL
LIN {X 0,Y 284.342,Z 348.685,A -85,B 0,C 180,E1 -17070.374,E2 -17070.374} C_VEL
LIN {X 0,Y 284.315,Z 348.687,A -85,B 0,C 180,E1 -17073.581,E2 -17073.581} C_VEL
LIN {X 0,Y 284.333,Z 348.688,A -85,B 0,C 180,E1 -17076.704,E2 -17076.704} C_VEL
LIN {X 0,Y 284.406,Z 348.678,A -85,B 0,C 180,E1 -17081.262,E2 -17081.262} C_VEL
LIN {X 0,Y 284.495,Z 348.673,A -85,B 0,C 180,E1 -17084.459,E2 -17084.459} C_VEL
LIN {X 0,Y 284.49,Z 348.673,A -85,B 0,C 180,E1 -17088.602,E2 -17088.602} C_VEL
LIN {X 0,Y 284.611,Z 348.646,A -85,B 0,C 180,E1 -17091.48,E2 -17091.48} C_VEL
LIN {X 0,Y 284.573,Z 348.663,A -85,B 0,C 180,E1 -17094.331,E2 -17094.331} C_VEL
LIN {X 0,Y 284.849,Z 348.628,A -85,B 0,C 180,E1 -17098.587,E2 -17098.587} C_VEL
LIN {X 0,Y 284.845,Z 348.617,A -85,B 0,C 180,E1 -17101.414,E2 -17101.414} C_VEL
LIN {X 0,Y 284.646,Z 348.639,A -85,B 0,C 180,E1 -17107.092,E2 -17107.092} C_VEL
LIN {X 0,Y 284.517,Z 348.667,A -85,B 0,C 180,E1 -17109.958,E2 -17109.958} C_VEL
LIN {X 0,Y 284.422,Z 348.681,A -85,B 0,C 180,E1 -17114.306,E2 -17114.306} C_VEL
LIN {X 0,Y 284.319,Z 348.694,A -85,B 0,C 180,E1 -17118.745,E2 -17118.745} C_VEL
LIN {X 0,Y 284.299,Z 348.69,A -85,B 0,C 180,E1 -17121.766,E2 -17121.766} C_VEL
LIN {X 0,Y 284.286,Z 348.689,A -85,B 0,C 180,E1 -17124.852,E2 -17124.852} C_VEL
LIN {X 0,Y 284.262,Z 348.694,A -85,B 0,C 180,E1 -17128.019,E2 -17128.019} C_VEL
LIN {X 0,Y 284.28,Z 348.669,A -85,B 0,C 180,E1 -17131.277,E2 -17131.277} C_VEL
LIN {X 0,Y 284.339,Z 348.673,A -85,B 0,C 180,E1 -17135.347,E2 -17135.347} C_VEL
LIN {X 0,Y 284.301,Z 348.685,A -85,B 0,C 180,E1 -17138.172,E2 -17138.172} C_VEL
LIN {X 0,Y 284.239,Z 348.704,A -85,B 0,C 180,E1 -17142.117,E2 -17142.117} C_VEL
LIN {X 0,Y 284.268,Z 348.69,A -85,B 0,C 180,E1 -17146.512,E2 -17146.512} C_VEL
LIN {X 0,Y 284.272,Z 348.84,A -85,B 0,C 180,E1 -17146.736,E2 -17146.736} C_VEL
LIN {X 0,Y 285.034,Z 351.319,A -85,B 0,C 180,E1 -17147.707,E2 -17147.707} C_VEL
LIN {X 0,Y 295.432,Z 369.332,A -85,B 0,C 180,E1 -17149.905,E2 -17149.905} C_VEL
LIN {X 0,Y 302.448,Z 383.082,A -85,B 0,C 180,E1 -17151.315,E2 -17151.315} C_VEL
LIN {X 0,Y 308.871,Z 397.295,A -85,B 0,C 180,E1 -17152.573,E2 -17152.573} C_VEL
LIN {X 0,Y 309.536,Z 398.76,A -85,B 0,C 180,E1 -17152.699,E2 -17152.699} C_VEL
LIN {X 0,Y 306.301,Z 486.916,A -85,B 0,C 180,E1 -17154.756,E2 -17154.756} C_VEL
LIN {X 0,Y 305.271,Z 500.807,A -85,B 0,C 180,E1 -17155.314,E2 -17155.314} C_VEL
LIN {X 0,Y 303.553,Z 515.105,A -85,B 0,C 180,E1 -17156.144,E2 -17156.144} C_VEL
LIN {X 0,Y 301.684,Z 527.833,A -85,B 0,C 180,E1 -17157.152,E2 -17157.152} C_VEL
LIN {X 0,Y 299.395,Z 541.043,A -85,B 0,C 180,E1 -17158.513,E2 -17158.513} C_VEL
LIN {X 0,Y 296.962,Z 552.603,A -85,B 0,C 180,E1 -17160.003,E2 -17160.003} C_VEL
LIN {X 0,Y 294.772,Z 562.206,A -85,B 0,C 180,E1 -17161.52,E2 -17161.52} C_VEL
LIN {X 0,Y 292.282,Z 572.86,A -85,B 0,C 180,E1 -17163.587,E2 -17163.587} C_VEL
LIN {X 0,Y 289.939,Z 581.619,A -85,B 0,C 180,E1 -17165.665,E2 -17165.665} C_VEL
LIN {X 0,Y 287.966,Z 588.88,A -85,B 0,C 180,E1 -17167.773,E2 -17167.773} C_VEL
LIN {X 0,Y 286.385,Z 594.896,A -85,B 0,C 180,E1 -17169.906,E2 -17169.906} C_VEL
LIN {X 0,Y 284.698,Z 601.281,A -85,B 0,C 180,E1 -17172.769,E2 -17172.769} C_VEL
LIN {X 0,Y 283.549,Z 606.013,A -85,B 0,C 180,E1 -17175.649,E2 -17175.649} C_VEL
LIN {X 0,Y 282.7,Z 609.221,A -85,B 0,C 180,E1 -17178.528,E2 -17178.528} C_VEL
LIN {X 0,Y 282.388,Z 611.026,A -85,B 0,C 180,E1 -17181.412,E2 -17181.412} C_VEL
LIN {X 0,Y 282.377,Z 611.499,A -85,B 0,C 180,E1 -17184.286,E2 -17184.286} C_VEL
LIN {X 0,Y 282.387,Z 610.662,A -85,B 0,C 180,E1 -17187.147,E2 -17187.147} C_VEL
LIN {X 0,Y 282.444,Z 608.506,A -85,B 0,C 180,E1 -17190,E2 -17190} C_VEL
LIN {X 0,Y 282.838,Z 604.974,A -85,B 0,C 180,E1 -17192.849,E2 -17192.849} C_VEL
LIN {X 0,Y 283.559,Z 601.365,A -85,B 0,C 180,E1 -17194.976,E2 -17194.976} C_VEL
LIN {X 0,Y 284.283,Z 596.848,A -85,B 0,C 180,E1 -17197.1,E2 -17197.1} C_VEL
LIN {X 0,Y 285.584,Z 590.304,A -85,B 0,C 180,E1 -17199.562,E2 -17199.562} C_VEL
LIN {X 0,Y 286.945,Z 582.202,A -85,B 0,C 180,E1 -17202.016,E2 -17202.016} C_VEL
LIN {X 0,Y 288.778,Z 573.713,A -85,B 0,C 180,E1 -17204.086,E2 -17204.086} C_VEL
LIN {X 0,Y 290.796,Z 563.439,A -85,B 0,C 180,E1 -17206.137,E2 -17206.137} C_VEL
LIN {X 0,Y 292.79,Z 551.968,A -85,B 0,C 180,E1 -17208.002,E2 -17208.002} C_VEL
LIN {X 0,Y 294.672,Z 540.511,A -85,B 0,C 180,E1 -17209.506,E2 -17209.506} C_VEL
LIN {X 0,Y 296.53,Z 527.933,A -85,B 0,C 180,E1 -17210.825,E2 -17210.825} C_VEL
LIN {X 0,Y 298.049,Z 514.95,A -85,B 0,C 180,E1 -17211.892,E2 -17211.892} C_VEL
LIN {X 0,Y 299.388,Z 500.927,A -85,B 0,C 180,E1 -17212.743,E2 -17212.743} C_VEL
LIN {X 0,Y 300.198,Z 487.293,A -85,B 0,C 180,E1 -17213.316,E2 -17213.316} C_VEL
LIN {X 0,Y 303.267,Z 393.198,A -85,B 0,C 180,E1 -17215.532,E2 -17215.532} C_VEL
LIN {X 0,Y 302.062,Z 389.328,A -85,B 0,C 180,E1 -17215.759,E2 -17215.759} C_VEL
LIN {X 0,Y 295.394,Z 372.928,A -85,B 0,C 180,E1 -17216.923,E2 -17216.923} C_VEL
LIN {X 0,Y 286.295,Z 353.667,A -85,B 0,C 180,E1 -17218.532,E2 -17218.532} C_VEL
LIN {X 0,Y 284.768,Z 350.437,A -85,B 0,C 180,E1 -17218.849,E2 -17218.849} C_VEL
LIN {X 0,Y 284.297,Z 348.691,A -85,B 0,C 180,E1 -17219.557,E2 -17219.557} C_VEL
LIN {X 0,Y 284.307,Z 348.695,A -85,B 0,C 180,E1 -17222.945,E2 -17222.945} C_VEL
LIN {X 0,Y 284.321,Z 348.693,A -85,B 0,C 180,E1 -17226.388,E2 -17226.388} C_VEL
LIN {X 0,Y 284.284,Z 348.697,A -85,B 0,C 180,E1 -17229.999,E2 -17229.999} C_VEL
LIN {X 0,Y 284.236,Z 348.704,A -85,B 0,C 180,E1 -17234.188,E2 -17234.188} C_VEL
LIN {X 0,Y 284.242,Z 348.699,A -85,B 0,C 180,E1 -17238.118,E2 -17238.118} C_VEL
LIN {X 0,Y 284.253,Z 348.696,A -85,B 0,C 180,E1 -17240.695,E2 -17240.695} C_VEL
LIN {X 0,Y 283.588,Z 348.782,A -85,B 0,C 180,E1 -17241.877,E2 -17241.877} C_VEL
LIN {X 0,Y 280.777,Z 349.131,A -85,B 0,C 180,E1 -17243.805,E2 -17243.805} C_VEL
LIN {X 0,Y 278.384,Z 349.432,A -85,B 0,C 180,E1 -17245.37,E2 -17245.37} C_VEL
LIN {X 0,Y 277.339,Z 349.555,A -85,B 0,C 180,E1 -17246.582,E2 -17246.582} C_VEL
LIN {X 0,Y 277.244,Z 349.564,A -85,B 0,C 180,E1 -17246.993,E2 -17246.993} C_VEL
LIN {X 0,Y 277.219,Z 349.573,A -85,B 0,C 180,E1 -17251.204,E2 -17251.204} C_VEL
LIN {X 0,Y 277.239,Z 349.574,A -85,B 0,C 180,E1 -17254.472,E2 -17254.472} C_VEL
LIN {X 0,Y 277.257,Z 349.559,A -85,B 0,C 180,E1 -17257.652,E2 -17257.652} C_VEL
LIN {X 0,Y 277.282,Z 349.542,A -85,B 0,C 180,E1 -17260.761,E2 -17260.761} C_VEL
LIN {X 0,Y 277.384,Z 349.555,A -85,B 0,C 180,E1 -17265.323,E2 -17265.323} C_VEL
LIN {X 0,Y 277.457,Z 349.513,A -85,B 0,C 180,E1 -17269.786,E2 -17269.786} C_VEL
LIN {X 0,Y 277.604,Z 349.53,A -85,B 0,C 180,E1 -17272.727,E2 -17272.727} C_VEL
LIN {X 0,Y 277.811,Z 349.505,A -85,B 0,C 180,E1 -17278.55,E2 -17278.55} C_VEL
LIN {X 0,Y 277.814,Z 349.495,A -85,B 0,C 180,E1 -17281.449,E2 -17281.449} C_VEL
LIN {X 0,Y 277.604,Z 349.528,A -85,B 0,C 180,E1 -17287.272,E2 -17287.272} C_VEL
LIN {X 0,Y 277.46,Z 349.543,A -85,B 0,C 180,E1 -17290.213,E2 -17290.213} C_VEL
LIN {X 0,Y 277.437,Z 349.546,A -85,B 0,C 180,E1 -17294.674,E2 -17294.674} C_VEL
LIN {X 0,Y 277.347,Z 349.559,A -85,B 0,C 180,E1 -17299.233,E2 -17299.233} C_VEL
LIN {X 0,Y 277.293,Z 349.572,A -85,B 0,C 180,E1 -17303.923,E2 -17303.923} C_VEL
LIN {X 0,Y 277.308,Z 349.57,A -85,B 0,C 180,E1 -17307.497,E2 -17307.497} C_VEL
LIN {X 0,Y 277.248,Z 349.577,A -85,B 0,C 180,E1 -17310.472,E2 -17310.472} C_VEL
LIN {X 0,Y 277.255,Z 349.579,A -85,B 0,C 180,E1 -17313.894,E2 -17313.894} C_VEL
LIN {X 0,Y 277.283,Z 349.575,A -85,B 0,C 180,E1 -17317.467,E2 -17317.467} C_VEL
LIN {X 0,Y 277.21,Z 349.583,A -85,B 0,C 180,E1 -17321.236,E2 -17321.236} C_VEL
LIN {X 0,Y 277.201,Z 349.583,A -85,B 0,C 180,E1 -17325.226,E2 -17325.226} C_VEL
LIN {X 0,Y 277.223,Z 349.579,A -85,B 0,C 180,E1 -17329.512,E2 -17329.512} C_VEL
LIN {X 0,Y 277.34,Z 349.745,A -85,B 0,C 180,E1 -17330.916,E2 -17330.916} C_VEL
LIN {X 0,Y 280.166,Z 360.749,A -85,B 0,C 180,E1 -17334.763,E2 -17334.763} C_VEL
LIN {X 0,Y 280.838,Z 363.866,A -85,B 0,C 180,E1 -17335.723,E2 -17335.723} C_VEL
LIN {X 0,Y 289.773,Z 383.897,A -85,B 0,C 180,E1 -17337.382,E2 -17337.382} C_VEL
LIN {X 0,Y 293.108,Z 392.755,A -85,B 0,C 180,E1 -17338.007,E2 -17338.007} C_VEL
LIN {X 0,Y 296.336,Z 414.501,A -85,B 0,C 180,E1 -17338.953,E2 -17338.953} C_VEL
LIN {X 0,Y 293.635,Z 501.519,A -85,B 0,C 180,E1 -17341.058,E2 -17341.058} C_VEL
LIN {X 0,Y 292.563,Z 515.599,A -85,B 0,C 180,E1 -17341.628,E2 -17341.628} C_VEL
LIN {X 0,Y 291.021,Z 529.882,A -85,B 0,C 180,E1 -17342.493,E2 -17342.493} C_VEL
LIN {X 0,Y 289.049,Z 543.96,A -85,B 0,C 180,E1 -17343.657,E2 -17343.657} C_VEL
LIN {X 0,Y 287.035,Z 557.059,A -85,B 0,C 180,E1 -17345.084,E2 -17345.084} C_VEL
LIN {X 0,Y 284.846,Z 569.218,A -85,B 0,C 180,E1 -17346.748,E2 -17346.748} C_VEL
LIN {X 0,Y 282.767,Z 579.56,A -85,B 0,C 180,E1 -17348.494,E2 -17348.494} C_VEL
LIN {X 0,Y 280.7,Z 589.837,A -85,B 0,C 180,E1 -17350.625,E2 -17350.625} C_VEL
LIN {X 0,Y 278.982,Z 598.226,A -85,B 0,C 180,E1 -17352.745,E2 -17352.745} C_VEL
LIN {X 0,Y 277.796,Z 605.453,A -85,B 0,C 180,E1 -17354.97,E2 -17354.97} C_VEL
LIN {X 0,Y 276.556,Z 612.207,A -85,B 0,C 180,E1 -17357.525,E2 -17357.525} C_VEL
LIN {X 0,Y 275.724,Z 618.195,A -85,B 0,C 180,E1 -17360.463,E2 -17360.463} C_VEL
LIN {X 0,Y 275.448,Z 621.657,A -85,B 0,C 180,E1 -17362.671,E2 -17362.671} C_VEL
LIN {X 0,Y 275.249,Z 624.937,A -85,B 0,C 180,E1 -17365.607,E2 -17365.607} C_VEL
LIN {X 0,Y 275.264,Z 626.804,A -85,B 0,C 180,E1 -17368.537,E2 -17368.537} C_VEL
LIN {X 0,Y 275.259,Z 627.318,A -85,B 0,C 180,E1 -17371.463,E2 -17371.463} C_VEL
LIN {X 0,Y 275.214,Z 626.495,A -85,B 0,C 180,E1 -17374.394,E2 -17374.394} C_VEL
LIN {X 0,Y 275.424,Z 624.332,A -85,B 0,C 180,E1 -17377.33,E2 -17377.33} C_VEL
LIN {X 0,Y 275.988,Z 620.78,A -85,B 0,C 180,E1 -17380.268,E2 -17380.268} C_VEL
LIN {X 0,Y 277.091,Z 615.74,A -85,B 0,C 180,E1 -17383.195,E2 -17383.195} C_VEL
LIN {X 0,Y 278.289,Z 610.886,A -85,B 0,C 180,E1 -17385.377,E2 -17385.377} C_VEL
LIN {X 0,Y 280.046,Z 603.907,A -85,B 0,C 180,E1 -17387.904,E2 -17387.904} C_VEL
LIN {X 0,Y 282.403,Z 595.279,A -85,B 0,C 180,E1 -17390.39,E2 -17390.39} C_VEL
LIN {X 0,Y 284.83,Z 586.281,A -85,B 0,C 180,E1 -17392.486,E2 -17392.486} C_VEL
LIN {X 0,Y 287.709,Z 575.402,A -85,B 0,C 180,E1 -17394.536,E2 -17394.536} C_VEL
LIN {X 0,Y 290.207,Z 565.059,A -85,B 0,C 180,E1 -17396.117,E2 -17396.117} C_VEL
LIN {X 0,Y 292.543,Z 553.72,A -85,B 0,C 180,E1 -17397.546,E2 -17397.546} C_VEL
LIN {X 0,Y 294.964,Z 540.662,A -85,B 0,C 180,E1 -17398.848,E2 -17398.848} C_VEL
LIN {X 0,Y 297.182,Z 526.897,A -85,B 0,C 180,E1 -17399.875,E2 -17399.875} C_VEL
LIN {X 0,Y 298.921,Z 512.323,A -85,B 0,C 180,E1 -17400.657,E2 -17400.657} C_VEL
LIN {X 0,Y 300.03,Z 497.14,A -85,B 0,C 180,E1 -17401.19,E2 -17401.19} C_VEL
LIN {X 0,Y 303.069,Z 417.558,A -85,B 0,C 180,E1 -17403.055,E2 -17403.055} C_VEL
LIN {X 0,Y 300.401,Z 402.093,A -85,B 0,C 180,E1 -17403.857,E2 -17403.857} C_VEL
LIN {X 0,Y 292.432,Z 384.539,A -85,B 0,C 180,E1 -17405.523,E2 -17405.523} C_VEL
LIN {X 0,Y 285.055,Z 370.497,A -85,B 0,C 180,E1 -17407.115,E2 -17407.115} C_VEL
LIN {X 0,Y 282.806,Z 366.465,A -85,B 0,C 180,E1 -17407.616,E2 -17407.616} C_VEL
LIN {X 0,Y 281.105,Z 362.976,A -85,B 0,C 180,E1 -17408.045,E2 -17408.045} C_VEL
LIN {X 0,Y 278.684,Z 354.566,A -85,B 0,C 180,E1 -17411.358,E2 -17411.358} C_VEL
LIN {X 0,Y 277.215,Z 349.575,A -85,B 0,C 180,E1 -17413.492,E2 -17413.492} C_VEL
LIN {X 0,Y 277.216,Z 349.576,A -85,B 0,C 180,E1 -17417.326,E2 -17417.326} C_VEL
LIN {X 0,Y 277.277,Z 349.569,A -85,B 0,C 180,E1 -17421.79,E2 -17421.79} C_VEL
LIN {X 0,Y 277.305,Z 349.563,A -85,B 0,C 180,E1 -17424.345,E2 -17424.345} C_VEL
LIN {X 0,Y 277.241,Z 349.573,A -85,B 0,C 180,E1 -17427.836,E2 -17427.836} C_VEL
LIN {X 0,Y 277.245,Z 349.573,A -85,B 0,C 180,E1 -17431.208,E2 -17431.208} C_VEL
LIN {X 0,Y 277.256,Z 349.567,A -85,B 0,C 180,E1 -17434.474,E2 -17434.474} C_VEL
LIN {X 0,Y 277.269,Z 349.562,A -85,B 0,C 180,E1 -17437.654,E2 -17437.654} C_VEL
LIN {X 0,Y 277.347,Z 349.559,A -85,B 0,C 180,E1 -17440.767,E2 -17440.767} C_VEL
LIN {X 0,Y 277.437,Z 349.55,A -85,B 0,C 180,E1 -17445.326,E2 -17445.326} C_VEL
LIN {X 0,Y 277.463,Z 349.548,A -85,B 0,C 180,E1 -17449.787,E2 -17449.787} C_VEL
LIN {X 0,Y 277.604,Z 349.523,A -85,B 0,C 180,E1 -17452.728,E2 -17452.728} C_VEL
LIN {X 0,Y 277.815,Z 349.504,A -85,B 0,C 180,E1 -17458.551,E2 -17458.551} C_VEL
LIN {X 0,Y 277.812,Z 349.492,A -85,B 0,C 180,E1 -17461.45,E2 -17461.45} C_VEL
LIN {X 0,Y 277.604,Z 349.516,A -85,B 0,C 180,E1 -17467.273,E2 -17467.273} C_VEL
LIN {X 0,Y 277.458,Z 349.545,A -85,B 0,C 180,E1 -17470.214,E2 -17470.214} C_VEL
LIN {X 0,Y 277.374,Z 349.558,A -85,B 0,C 180,E1 -17474.678,E2 -17474.678} C_VEL
LIN {X 0,Y 277.278,Z 349.571,A -85,B 0,C 180,E1 -17479.239,E2 -17479.239} C_VEL
LIN {X 0,Y 277.258,Z 349.568,A -85,B 0,C 180,E1 -17483.928,E2 -17483.928} C_VEL
LIN {X 0,Y 277.238,Z 349.573,A -85,B 0,C 180,E1 -17487.469,E2 -17487.469} C_VEL
LIN {X 0,Y 277.231,Z 349.542,A -85,B 0,C 180,E1 -17490.466,E2 -17490.466} C_VEL
LIN {X 0,Y 277.249,Z 349.575,A -85,B 0,C 180,E1 -17493.896,E2 -17493.896} C_VEL
LIN {X 0,Y 277.257,Z 349.552,A -85,B 0,C 180,E1 -17497.472,E2 -17497.472} C_VEL
LIN {X 0,Y 277.187,Z 349.582,A -85,B 0,C 180,E1 -17501.241,E2 -17501.241} C_VEL
LIN {X 0,Y 277.176,Z 349.572,A -85,B 0,C 180,E1 -17505.232,E2 -17505.232} C_VEL
LIN {X 0,Y 277.245,Z 349.816,A -85,B 0,C 180,E1 -17505.761,E2 -17505.761} C_VEL
LIN {X 0,Y 277.8,Z 351.609,A -85,B 0,C 180,E1 -17506.465,E2 -17506.465} C_VEL
LIN {X 0,Y 280.276,Z 355.647,A -85,B 0,C 180,E1 -17507.037,E2 -17507.037} C_VEL
LIN {X 0,Y 290.149,Z 372.636,A -85,B 0,C 180,E1 -17509.202,E2 -17509.202} C_VEL
LIN {X 0,Y 297.849,Z 387.881,A -85,B 0,C 180,E1 -17510.809,E2 -17510.809} C_VEL
LIN {X 0,Y 303.616,Z 400.871,A -85,B 0,C 180,E1 -17511.983,E2 -17511.983} C_VEL
LIN {X 0,Y 300.311,Z 487.787,A -85,B 0,C 180,E1 -17514.057,E2 -17514.057} C_VEL
LIN {X 0,Y 299.146,Z 502.081,A -85,B 0,C 180,E1 -17514.653,E2 -17514.653} C_VEL
LIN {X 0,Y 297.466,Z 515.532,A -85,B 0,C 180,E1 -17515.456,E2 -17515.456} C_VEL
LIN {X 0,Y 295.467,Z 528.557,A -85,B 0,C 180,E1 -17516.512,E2 -17516.512} C_VEL
LIN {X 0,Y 293.312,Z 540.669,A -85,B 0,C 180,E1 -17517.783,E2 -17517.783} C_VEL
LIN {X 0,Y 290.691,Z 552.327,A -85,B 0,C 180,E1 -17519.287,E2 -17519.287} C_VEL
LIN {X 0,Y 288.462,Z 562.014,A -85,B 0,C 180,E1 -17520.838,E2 -17520.838} C_VEL
LIN {X 0,Y 285.854,Z 572.733,A -85,B 0,C 180,E1 -17522.945,E2 -17522.945} C_VEL
LIN {X 0,Y 283.38,Z 581.548,A -85,B 0,C 180,E1 -17525.063,E2 -17525.063} C_VEL
LIN {X 0,Y 281.314,Z 588.858,A -85,B 0,C 180,E1 -17527.218,E2 -17527.218} C_VEL
LIN {X 0,Y 279.615,Z 594.917,A -85,B 0,C 180,E1 -17529.397,E2 -17529.397} C_VEL
LIN {X 0,Y 277.823,Z 601.34,A -85,B 0,C 180,E1 -17532.328,E2 -17532.328} C_VEL
LIN {X 0,Y 276.574,Z 606.109,A -85,B 0,C 180,E1 -17535.279,E2 -17535.279} C_VEL
LIN {X 0,Y 275.678,Z 609.364,A -85,B 0,C 180,E1 -17538.232,E2 -17538.232} C_VEL
LIN {X 0,Y 275.317,Z 611.204,A -85,B 0,C 180,E1 -17541.19,E2 -17541.19} C_VEL
LIN {X 0,Y 275.288,Z 611.71,A -85,B 0,C 180,E1 -17544.139,E2 -17544.139} C_VEL
LIN {X 0,Y 275.292,Z 610.904,A -85,B 0,C 180,E1 -17547.073,E2 -17547.073} C_VEL
LIN {X 0,Y 275.362,Z 608.78,A -85,B 0,C 180,E1 -17550,E2 -17550} C_VEL
LIN {X 0,Y 275.764,Z 605.282,A -85,B 0,C 180,E1 -17552.922,E2 -17552.922} C_VEL
LIN {X 0,Y 276.491,Z 601.71,A -85,B 0,C 180,E1 -17555.104,E2 -17555.104} C_VEL
LIN {X 0,Y 277.636,Z 595.482,A -85,B 0,C 180,E1 -17558.003,E2 -17558.003} C_VEL
LIN {X 0,Y 279.089,Z 588.195,A -85,B 0,C 180,E1 -17560.638,E2 -17560.638} C_VEL
LIN {X 0,Y 280.528,Z 579.993,A -85,B 0,C 180,E1 -17563.031,E2 -17563.031} C_VEL
LIN {X 0,Y 282.605,Z 571.011,A -85,B 0,C 180,E1 -17565.137,E2 -17565.137} C_VEL
LIN {X 0,Y 284.759,Z 560.161,A -85,B 0,C 180,E1 -17567.228,E2 -17567.228} C_VEL
LIN {X 0,Y 286.742,Z 549.137,A -85,B 0,C 180,E1 -17568.951,E2 -17568.951} C_VEL
LIN {X 0,Y 288.75,Z 536.973,A -85,B 0,C 180,E1 -17570.48,E2 -17570.48} C_VEL
LIN {X 0,Y 290.4,Z 525.308,A -85,B 0,C 180,E1 -17571.658,E2 -17571.658} C_VEL
LIN {X 0,Y 292.029,Z 511.351,A -85,B 0,C 180,E1 -17572.741,E2 -17572.741} C_VEL
LIN {X 0,Y 293.282,Z 497.363,A -85,B 0,C 180,E1 -17573.524,E2 -17573.524} C_VEL
LIN {X 0,Y 294.104,Z 483.299,A -85,B 0,C 180,E1 -17574.042,E2 -17574.042} C_VEL
LIN {X 0,Y 296.967,Z 394.279,A -85,B 0,C 180,E1 -17576.167,E2 -17576.167} C_VEL
LIN {X 0,Y 290.836,Z 378.595,A -85,B 0,C 180,E1 -17577.283,E2 -17577.283} C_VEL
LIN {X 0,Y 282.472,Z 360.61,A -85,B 0,C 180,E1 -17578.805,E2 -17578.805} C_VEL
LIN {X 0,Y 277.506,Z 350.718,A -85,B 0,C 180,E1 -17579.759,E2 -17579.759} C_VEL
LIN {X 0,Y 277.23,Z 349.569,A -85,B 0,C 180,E1 -17580.218,E2 -17580.218} C_VEL
LIN {X 0,Y 277.248,Z 349.575,A -85,B 0,C 180,E1 -17583.896,E2 -17583.896} C_VEL
LIN {X 0,Y 277.253,Z 349.574,A -85,B 0,C 180,E1 -17587.472,E2 -17587.472} C_VEL
LIN {X 0,Y 277.186,Z 349.58,A -85,B 0,C 180,E1 -17591.241,E2 -17591.241} C_VEL
LIN {X 0,Y 277.176,Z 349.578,A -85,B 0,C 180,E1 -17595.232,E2 -17595.232} C_VEL
LIN {X 0,Y 277.186,Z 349.576,A -85,B 0,C 180,E1 -17598.758,E2 -17598.758} C_VEL
LIN {X 0,Y 277.236,Z 349.569,A -85,B 0,C 180,E1 -17602.525,E2 -17602.525} C_VEL
LIN {X 0,Y 277.248,Z 349.571,A -85,B 0,C 180,E1 -17606.104,E2 -17606.104} C_VEL
LIN {X 0,Y 277.244,Z 349.564,A -85,B 0,C 180,E1 -17606.993,E2 -17606.993} C_VEL
LIN {X 0,Y 276.541,Z 349.655,A -85,B 0,C 180,E1 -17608.204,E2 -17608.204} C_VEL
LIN {X 0,Y 273.655,Z 350.024,A -85,B 0,C 180,E1 -17610.177,E2 -17610.177} C_VEL
LIN {X 0,Y 271.242,Z 350.315,A -85,B 0,C 180,E1 -17611.78,E2 -17611.78} C_VEL
LIN {X 0,Y 270.235,Z 350.437,A -85,B 0,C 180,E1 -17613.024,E2 -17613.024} C_VEL
LIN {X 0,Y 270.168,Z 350.447,A -85,B 0,C 180,E1 -17613.445,E2 -17613.445} C_VEL
LIN {X 0,Y 270.194,Z 350.446,A -85,B 0,C 180,E1 -17617.035,E2 -17617.035} C_VEL
LIN {X 0,Y 270.223,Z 350.417,A -85,B 0,C 180,E1 -17620.238,E2 -17620.238} C_VEL
LIN {X 0,Y 270.346,Z 350.432,A -85,B 0,C 180,E1 -17624.932,E2 -17624.932} C_VEL
LIN {X 0,Y 270.39,Z 350.391,A -85,B 0,C 180,E1 -17629.516,E2 -17629.516} C_VEL
LIN {X 0,Y 270.565,Z 350.403,A -85,B 0,C 180,E1 -17632.537,E2 -17632.537} C_VEL
LIN {X 0,Y 270.778,Z 350.381,A -85,B 0,C 180,E1 -17638.512,E2 -17638.512} C_VEL
LIN {X 0,Y 270.779,Z 350.372,A -85,B 0,C 180,E1 -17641.487,E2 -17641.487} C_VEL
LIN {X 0,Y 270.565,Z 350.406,A -85,B 0,C 180,E1 -17647.462,E2 -17647.462} C_VEL
LIN {X 0,Y 270.412,Z 350.421,A -85,B 0,C 180,E1 -17650.482,E2 -17650.482} C_VEL
LIN {X 0,Y 270.405,Z 350.422,A -85,B 0,C 180,E1 -17655.064,E2 -17655.064} C_VEL
LIN {X 0,Y 270.304,Z 350.44,A -85,B 0,C 180,E1 -17659.755,E2 -17659.755} C_VEL
LIN {X 0,Y 270.235,Z 350.448,A -85,B 0,C 180,E1 -17664.589,E2 -17664.589} C_VEL
LIN {X 0,Y 270.243,Z 350.449,A -85,B 0,C 180,E1 -17667.911,E2 -17667.911} C_VEL
LIN {X 0,Y 270.175,Z 350.46,A -85,B 0,C 180,E1 -17671.349,E2 -17671.349} C_VEL
LIN {X 0,Y 270.216,Z 350.454,A -85,B 0,C 180,E1 -17674.903,E2 -17674.903} C_VEL
LIN {X 0,Y 270.223,Z 350.449,A -85,B 0,C 180,E1 -17678.717,E2 -17678.717} C_VEL
LIN {X 0,Y 270.166,Z 350.46,A -85,B 0,C 180,E1 -17683.249,E2 -17683.249} C_VEL
LIN {X 0,Y 270.172,Z 350.456,A -85,B 0,C 180,E1 -17687.441,E2 -17687.441} C_VEL
LIN {X 0,Y 270.221,Z 350.497,A -85,B 0,C 180,E1 -17690.106,E2 -17690.106} C_VEL
LIN {X 0,Y 272.713,Z 360.221,A -85,B 0,C 180,E1 -17693.649,E2 -17693.649} C_VEL
LIN {X 0,Y 273.615,Z 363.547,A -85,B 0,C 180,E1 -17694.766,E2 -17694.766} C_VEL
LIN {X 0,Y 283.645,Z 385.929,A -85,B 0,C 180,E1 -17696.716,E2 -17696.716} C_VEL
LIN {X 0,Y 287.159,Z 395.228,A -85,B 0,C 180,E1 -17697.399,E2 -17697.399} C_VEL
LIN {X 0,Y 290.121,Z 415.528,A -85,B 0,C 180,E1 -17698.307,E2 -17698.307} C_VEL
LIN {X 0,Y 287.249,Z 502.276,A -85,B 0,C 180,E1 -17700.452,E2 -17700.452} C_VEL
LIN {X 0,Y 286.056,Z 516.781,A -85,B 0,C 180,E1 -17701.073,E2 -17701.073} C_VEL
LIN {X 0,Y 284.414,Z 531.276,A -85,B 0,C 180,E1 -17701.998,E2 -17701.998} C_VEL
LIN {X 0,Y 282.392,Z 545.007,A -85,B 0,C 180,E1 -17703.187,E2 -17703.187} C_VEL
LIN {X 0,Y 280.357,Z 557.646,A -85,B 0,C 180,E1 -17704.617,E2 -17704.617} C_VEL
LIN {X 0,Y 278.056,Z 569.796,A -85,B 0,C 180,E1 -17706.344,E2 -17706.344} C_VEL
LIN {X 0,Y 275.714,Z 580.911,A -85,B 0,C 180,E1 -17708.309,E2 -17708.309} C_VEL
LIN {X 0,Y 273.629,Z 590.912,A -85,B 0,C 180,E1 -17710.494,E2 -17710.494} C_VEL
LIN {X 0,Y 271.843,Z 599.456,A -85,B 0,C 180,E1 -17712.781,E2 -17712.781} C_VEL
LIN {X 0,Y 270.654,Z 606.129,A -85,B 0,C 180,E1 -17714.95,E2 -17714.95} C_VEL
LIN {X 0,Y 269.583,Z 611.878,A -85,B 0,C 180,E1 -17717.197,E2 -17717.197} C_VEL
LIN {X 0,Y 268.666,Z 617.899,A -85,B 0,C 180,E1 -17720.21,E2 -17720.21} C_VEL
LIN {X 0,Y 268.363,Z 621.375,A -85,B 0,C 180,E1 -17722.476,E2 -17722.476} C_VEL
LIN {X 0,Y 268.167,Z 624.69,A -85,B 0,C 180,E1 -17725.491,E2 -17725.491} C_VEL
LIN {X 0,Y 268.19,Z 626.585,A -85,B 0,C 180,E1 -17728.498,E2 -17728.498} C_VEL
LIN {X 0,Y 268.184,Z 627.123,A -85,B 0,C 180,E1 -17731.502,E2 -17731.502} C_VEL
LIN {X 0,Y 268.13,Z 626.323,A -85,B 0,C 180,E1 -17734.51,E2 -17734.51} C_VEL
LIN {X 0,Y 268.344,Z 624.184,A -85,B 0,C 180,E1 -17737.525,E2 -17737.525} C_VEL
LIN {X 0,Y 268.955,Z 620.656,A -85,B 0,C 180,E1 -17740.54,E2 -17740.54} C_VEL
LIN {X 0,Y 270.134,Z 615.644,A -85,B 0,C 180,E1 -17743.542,E2 -17743.542} C_VEL
LIN {X 0,Y 271.907,Z 609.003,A -85,B 0,C 180,E1 -17746.518,E2 -17746.518} C_VEL
LIN {X 0,Y 273.884,Z 601.632,A -85,B 0,C 180,E1 -17749.097,E2 -17749.097} C_VEL
LIN {X 0,Y 276.507,Z 592.49,A -85,B 0,C 180,E1 -17751.626,E2 -17751.626} C_VEL
LIN {X 0,Y 279.206,Z 582.951,A -85,B 0,C 180,E1 -17753.75,E2 -17753.75} C_VEL
LIN {X 0,Y 282.043,Z 572.398,A -85,B 0,C 180,E1 -17755.655,E2 -17755.655} C_VEL
LIN {X 0,Y 284.824,Z 560.576,A -85,B 0,C 180,E1 -17757.387,E2 -17757.387} C_VEL
LIN {X 0,Y 287.507,Z 547.834,A -85,B 0,C 180,E1 -17758.868,E2 -17758.868} C_VEL
LIN {X 0,Y 289.807,Z 535.162,A -85,B 0,C 180,E1 -17760.011,E2 -17760.011} C_VEL
LIN {X 0,Y 291.965,Z 520.977,A -85,B 0,C 180,E1 -17760.966,E2 -17760.966} C_VEL
LIN {X 0,Y 293.51,Z 506.61,A -85,B 0,C 180,E1 -17761.637,E2 -17761.637} C_VEL
LIN {X 0,Y 294.37,Z 491.916,A -85,B 0,C 180,E1 -17762.075,E2 -17762.075} C_VEL
LIN {X 0,Y 297.241,Z 418.213,A -85,B 0,C 180,E1 -17763.826,E2 -17763.826} C_VEL
LIN {X 0,Y 294.874,Z 404.943,A -85,B 0,C 180,E1 -17764.551,E2 -17764.551} C_VEL
LIN {X 0,Y 287.355,Z 388.272,A -85,B 0,C 180,E1 -17766.187,E2 -17766.187} C_VEL
LIN {X 0,Y 280.414,Z 374.866,A -85,B 0,C 180,E1 -17767.747,E2 -17767.747} C_VEL
LIN {X 0,Y 275.763,Z 366.539,A -85,B 0,C 180,E1 -17768.836,E2 -17768.836} C_VEL
LIN {X 0,Y 273.78,Z 362.737,A -85,B 0,C 180,E1 -17769.347,E2 -17769.347} C_VEL
LIN {X 0,Y 271.389,Z 354.594,A -85,B 0,C 180,E1 -17772.728,E2 -17772.728} C_VEL
LIN {X 0,Y 270.158,Z 350.459,A -85,B 0,C 180,E1 -17774.619,E2 -17774.619} C_VEL
LIN {X 0,Y 270.17,Z 350.453,A -85,B 0,C 180,E1 -17778.972,E2 -17778.972} C_VEL
LIN {X 0,Y 270.208,Z 350.446,A -85,B 0,C 180,E1 -17781.375,E2 -17781.375} C_VEL
LIN {X 0,Y 270.216,Z 350.451,A -85,B 0,C 180,E1 -17785.097,E2 -17785.097} C_VEL
LIN {X 0,Y 270.185,Z 350.453,A -85,B 0,C 180,E1 -17789.137,E2 -17789.137} C_VEL
LIN {X 0,Y 270.225,Z 350.451,A -85,B 0,C 180,E1 -17792.163,E2 -17792.163} C_VEL
LIN {X 0,Y 270.231,Z 350.448,A -85,B 0,C 180,E1 -17795.542,E2 -17795.542} C_VEL
LIN {X 0,Y 270.304,Z 350.44,A -85,B 0,C 180,E1 -17800.245,E2 -17800.245} C_VEL
LIN {X 0,Y 270.406,Z 350.426,A -85,B 0,C 180,E1 -17804.936,E2 -17804.936} C_VEL
LIN {X 0,Y 270.415,Z 350.427,A -85,B 0,C 180,E1 -17809.518,E2 -17809.518} C_VEL
LIN {X 0,Y 270.565,Z 350.398,A -85,B 0,C 180,E1 -17812.538,E2 -17812.538} C_VEL
LIN {X 0,Y 270.779,Z 350.38,A -85,B 0,C 180,E1 -17818.513,E2 -17818.513} C_VEL
LIN {X 0,Y 270.779,Z 350.368,A -85,B 0,C 180,E1 -17821.488,E2 -17821.488} C_VEL
LIN {X 0,Y 270.566,Z 350.394,A -85,B 0,C 180,E1 -17827.463,E2 -17827.463} C_VEL
LIN {X 0,Y 270.409,Z 350.422,A -85,B 0,C 180,E1 -17830.483,E2 -17830.483} C_VEL
LIN {X 0,Y 270.341,Z 350.432,A -85,B 0,C 180,E1 -17835.069,E2 -17835.069} C_VEL
LIN {X 0,Y 270.222,Z 350.444,A -85,B 0,C 180,E1 -17839.762,E2 -17839.762} C_VEL
LIN {X 0,Y 270.185,Z 350.446,A -85,B 0,C 180,E1 -17844.436,E2 -17844.436} C_VEL
LIN {X 0,Y 270.187,Z 350.447,A -85,B 0,C 180,E1 -17847.919,E2 -17847.919} C_VEL
LIN {X 0,Y 270.171,Z 350.426,A -85,B 0,C 180,E1 -17851.351,E2 -17851.351} C_VEL
LIN {X 0,Y 270.201,Z 350.439,A -85,B 0,C 180,E1 -17854.906,E2 -17854.906} C_VEL
LIN {X 0,Y 270.201,Z 350.451,A -85,B 0,C 180,E1 -17858.711,E2 -17858.711} C_VEL
LIN {X 0,Y 270.151,Z 350.458,A -85,B 0,C 180,E1 -17863.245,E2 -17863.245} C_VEL
LIN {X 0,Y 270.164,Z 350.566,A -85,B 0,C 180,E1 -17864.619,E2 -17864.619} C_VEL
LIN {X 0,Y 270.457,Z 351.842,A -85,B 0,C 180,E1 -17865.108,E2 -17865.108} C_VEL
LIN {X 0,Y 272.368,Z 355.014,A -85,B 0,C 180,E1 -17865.583,E2 -17865.583} C_VEL
LIN {X 0,Y 274.153,Z 357.771,A -85,B 0,C 180,E1 -17866.011,E2 -17866.011} C_VEL
LIN {X 0,Y 279.738,Z 366.948,A -85,B 0,C 180,E1 -17867.316,E2 -17867.316} C_VEL
LIN {X 0,Y 287.188,Z 380.38,A -85,B 0,C 180,E1 -17868.979,E2 -17868.979} C_VEL
LIN {X 0,Y 294.52,Z 395.383,A -85,B 0,C 180,E1 -17870.551,E2 -17870.551} C_VEL
LIN {X 0,Y 297.749,Z 402.84,A -85,B 0,C 180,E1 -17871.234,E2 -17871.234} C_VEL
LIN {X 0,Y 294.448,Z 487.345,A -85,B 0,C 180,E1 -17873.281,E2 -17873.281} C_VEL
LIN {X 0,Y 293.262,Z 501.834,A -85,B 0,C 180,E1 -17873.886,E2 -17873.886} C_VEL
LIN {X 0,Y 291.455,Z 515.844,A -85,B 0,C 180,E1 -17874.733,E2 -17874.733} C_VEL
LIN {X 0,Y 289.292,Z 529.276,A -85,B 0,C 180,E1 -17875.844,E2 -17875.844} C_VEL
LIN {X 0,Y 286.959,Z 541.733,A -85,B 0,C 180,E1 -17877.189,E2 -17877.189} C_VEL
LIN {X 0,Y 284.257,Z 553.237,A -85,B 0,C 180,E1 -17878.721,E2 -17878.721} C_VEL
LIN {X 0,Y 281.709,Z 563.791,A -85,B 0,C 180,E1 -17880.482,E2 -17880.482} C_VEL
LIN {X 0,Y 278.995,Z 574.242,A -85,B 0,C 180,E1 -17882.63,E2 -17882.63} C_VEL
LIN {X 0,Y 276.452,Z 582.835,A -85,B 0,C 180,E1 -17884.797,E2 -17884.797} C_VEL
LIN {X 0,Y 273.902,Z 591.308,A -85,B 0,C 180,E1 -17887.477,E2 -17887.477} C_VEL
LIN {X 0,Y 272.334,Z 596.748,A -85,B 0,C 180,E1 -17889.611,E2 -17889.611} C_VEL
LIN {X 0,Y 270.962,Z 601.4,A -85,B 0,C 180,E1 -17891.865,E2 -17891.865} C_VEL
LIN {X 0,Y 269.624,Z 606.205,A -85,B 0,C 180,E1 -17894.891,E2 -17894.891} C_VEL
LIN {X 0,Y 268.668,Z 609.502,A -85,B 0,C 180,E1 -17897.92,E2 -17897.92} C_VEL
LIN {X 0,Y 268.26,Z 611.383,A -85,B 0,C 180,E1 -17900.956,E2 -17900.956} C_VEL
LIN {X 0,Y 268.206,Z 611.92,A -85,B 0,C 180,E1 -17903.983,E2 -17903.983} C_VEL
LIN {X 0,Y 268.2,Z 611.146,A -85,B 0,C 180,E1 -17906.996,E2 -17906.996} C_VEL
LIN {X 0,Y 268.281,Z 609.053,A -85,B 0,C 180,E1 -17910,E2 -17910} C_VEL
LIN {X 0,Y 268.693,Z 605.589,A -85,B 0,C 180,E1 -17912.999,E2 -17912.999} C_VEL
LIN {X 0,Y 269.613,Z 600.645,A -85,B 0,C 180,E1 -17915.985,E2 -17915.985} C_VEL
LIN {X 0,Y 271.011,Z 594.069,A -85,B 0,C 180,E1 -17918.951,E2 -17918.951} C_VEL
LIN {X 0,Y 272.447,Z 586.868,A -85,B 0,C 180,E1 -17921.498,E2 -17921.498} C_VEL
LIN {X 0,Y 273.996,Z 579.118,A -85,B 0,C 180,E1 -17923.725,E2 -17923.725} C_VEL
LIN {X 0,Y 276.194,Z 569.916,A -85,B 0,C 180,E1 -17925.875,E2 -17925.875} C_VEL
LIN {X 0,Y 278.225,Z 559.768,A -85,B 0,C 180,E1 -17927.835,E2 -17927.835} C_VEL
LIN {X 0,Y 280.257,Z 548.596,A -85,B 0,C 180,E1 -17929.597,E2 -17929.597} C_VEL
LIN {X 0,Y 282.163,Z 537.788,A -85,B 0,C 180,E1 -17930.98,E2 -17930.98} C_VEL
LIN {X 0,Y 284.1,Z 524.335,A -85,B 0,C 180,E1 -17932.355,E2 -17932.355} C_VEL
LIN {X 0,Y 285.694,Z 511.293,A -85,B 0,C 180,E1 -17933.37,E2 -17933.37} C_VEL
LIN {X 0,Y 286.989,Z 497.2,A -85,B 0,C 180,E1 -17934.169,E2 -17934.169} C_VEL
LIN {X 0,Y 287.808,Z 483.427,A -85,B 0,C 180,E1 -17934.682,E2 -17934.682} C_VEL
LIN {X 0,Y 290.707,Z 395.868,A -85,B 0,C 180,E1 -17936.814,E2 -17936.814} C_VEL
LIN {X 0,Y 284.645,Z 380.571,A -85,B 0,C 180,E1 -17937.957,E2 -17937.957} C_VEL
LIN {X 0,Y 275.724,Z 361.38,A -85,B 0,C 180,E1 -17939.655,E2 -17939.655} C_VEL
LIN {X 0,Y 271.604,Z 353.863,A -85,B 0,C 180,E1 -17940.447,E2 -17940.447} C_VEL
LIN {X 0,Y 270.367,Z 351.41,A -85,B 0,C 180,E1 -17940.697,E2 -17940.697} C_VEL
LIN {X 0,Y 270.215,Z 350.614,A -85,B 0,C 180,E1 -17940.873,E2 -17940.873} C_VEL
LIN {X 0,Y 270.2,Z 350.451,A -85,B 0,C 180,E1 -17944.906,E2 -17944.906} C_VEL
LIN {X 0,Y 270.201,Z 350.451,A -85,B 0,C 180,E1 -17948.71,E2 -17948.71} C_VEL
LIN {X 0,Y 270.15,Z 350.46,A -85,B 0,C 180,E1 -17953.245,E2 -17953.245} C_VEL
LIN {X 0,Y 270.153,Z 350.457,A -85,B 0,C 180,E1 -17957.437,E2 -17957.437} C_VEL
LIN {X 0,Y 270.173,Z 350.454,A -85,B 0,C 180,E1 -17961.368,E2 -17961.368} C_VEL
LIN {X 0,Y 270.2,Z 350.452,A -85,B 0,C 180,E1 -17965.094,E2 -17965.094} C_VEL
LIN {X 0,Y 270.173,Z 350.456,A -85,B 0,C 180,E1 -17969.141,E2 -17969.141} C_VEL
LIN {X 0,Y 270.168,Z 350.447,A -85,B 0,C 180,E1 -17973.445,E2 -17973.445} C_VEL
LIN {X 0,Y 269.553,Z 350.534,A -85,B 0,C 180,E1 -17974.688,E2 -17974.688} C_VEL
LIN {X 0,Y 266.769,Z 350.874,A -85,B 0,C 180,E1 -17976.716,E2 -17976.716} C_VEL
LIN {X 0,Y 264.357,Z 351.155,A -85,B 0,C 180,E1 -17978.364,E2 -17978.364} C_VEL
LIN {X 0,Y 263.285,Z 351.279,A -85,B 0,C 180,E1 -17979.641,E2 -17979.641} C_VEL
LIN {X 0,Y 263.18,Z 351.293,A -85,B 0,C 180,E1 -17980.074,E2 -17980.074} C_VEL
LIN {X 0,Y 263.293,Z 351.313,A -85,B 0,C 180,E1 -17984.518,E2 -17984.518} C_VEL
LIN {X 0,Y 263.335,Z 351.268,A -85,B 0,C 180,E1 -17989.232,E2 -17989.232} C_VEL
LIN {X 0,Y 263.529,Z 351.277,A -85,B 0,C 180,E1 -17992.337,E2 -17992.337} C_VEL
LIN {X 0,Y 263.743,Z 351.258,A -85,B 0,C 180,E1 -17998.473,E2 -17998.473} C_VEL
LIN {X 0,Y 263.742,Z 351.248,A -85,B 0,C 180,E1 -18001.527,E2 -18001.527} C_VEL
LIN {X 0,Y 263.529,Z 351.284,A -85,B 0,C 180,E1 -18007.662,E2 -18007.662} C_VEL
LIN {X 0,Y 263.355,Z 351.301,A -85,B 0,C 180,E1 -18010.766,E2 -18010.766} C_VEL
LIN {X 0,Y 263.353,Z 351.302,A -85,B 0,C 180,E1 -18015.477,E2 -18015.477} C_VEL
LIN {X 0,Y 263.265,Z 351.317,A -85,B 0,C 180,E1 -18020.306,E2 -18020.306} C_VEL
LIN {X 0,Y 263.187,Z 351.324,A -85,B 0,C 180,E1 -18025.293,E2 -18025.293} C_VEL
LIN {X 0,Y 263.154,Z 351.329,A -85,B 0,C 180,E1 -18028.732,E2 -18028.732} C_VEL
LIN {X 0,Y 263.13,Z 351.331,A -85,B 0,C 180,E1 -18032.288,E2 -18032.288} C_VEL
LIN {X 0,Y 263.189,Z 351.327,A -85,B 0,C 180,E1 -18035.977,E2 -18035.977} C_VEL
LIN {X 0,Y 263.116,Z 351.34,A -85,B 0,C 180,E1 -18039.87,E2 -18039.87} C_VEL
LIN {X 0,Y 263.123,Z 351.336,A -85,B 0,C 180,E1 -18043.984,E2 -18043.984} C_VEL
LIN {X 0,Y 263.125,Z 351.333,A -85,B 0,C 180,E1 -18048.406,E2 -18048.406} C_VEL
LIN {X 0,Y 263.158,Z 351.486,A -85,B 0,C 180,E1 -18049.335,E2 -18049.335} C_VEL
LIN {X 0,Y 265.439,Z 360.029,A -85,B 0,C 180,E1 -18052.589,E2 -18052.589} C_VEL
LIN {X 0,Y 266.208,Z 363.16,A -85,B 0,C 180,E1 -18053.719,E2 -18053.719} C_VEL
LIN {X 0,Y 274.552,Z 381.068,A -85,B 0,C 180,E1 -18055.425,E2 -18055.425} C_VEL
LIN {X 0,Y 280.602,Z 395.697,A -85,B 0,C 180,E1 -18056.629,E2 -18056.629} C_VEL
LIN {X 0,Y 281.355,Z 398.469,A -85,B 0,C 180,E1 -18056.802,E2 -18056.802} C_VEL
LIN {X 0,Y 283.964,Z 417.381,A -85,B 0,C 180,E1 -18057.659,E2 -18057.659} C_VEL
LIN {X 0,Y 280.992,Z 501.846,A -85,B 0,C 180,E1 -18059.778,E2 -18059.778} C_VEL
LIN {X 0,Y 279.746,Z 516.425,A -85,B 0,C 180,E1 -18060.408,E2 -18060.408} C_VEL
LIN {X 0,Y 278.126,Z 530.394,A -85,B 0,C 180,E1 -18061.307,E2 -18061.307} C_VEL
LIN {X 0,Y 276.031,Z 544.273,A -85,B 0,C 180,E1 -18062.517,E2 -18062.517} C_VEL
LIN {X 0,Y 273.934,Z 556.873,A -85,B 0,C 180,E1 -18063.958,E2 -18063.958} C_VEL
LIN {X 0,Y 271.534,Z 569.271,A -85,B 0,C 180,E1 -18065.739,E2 -18065.739} C_VEL
LIN {X 0,Y 269.088,Z 580.442,A -85,B 0,C 180,E1 -18067.746,E2 -18067.746} C_VEL
LIN {X 0,Y 266.877,Z 590.485,A -85,B 0,C 180,E1 -18069.98,E2 -18069.98} C_VEL
LIN {X 0,Y 265.038,Z 598.82,A -85,B 0,C 180,E1 -18072.246,E2 -18072.246} C_VEL
LIN {X 0,Y 263.773,Z 605.776,A -85,B 0,C 180,E1 -18074.547,E2 -18074.547} C_VEL
LIN {X 0,Y 262.625,Z 611.546,A -85,B 0,C 180,E1 -18076.852,E2 -18076.852} C_VEL
LIN {X 0,Y 261.629,Z 617.603,A -85,B 0,C 180,E1 -18079.944,E2 -18079.944} C_VEL
LIN {X 0,Y 261.301,Z 621.094,A -85,B 0,C 180,E1 -18082.271,E2 -18082.271} C_VEL
LIN {X 0,Y 261.073,Z 624.44,A -85,B 0,C 180,E1 -18085.368,E2 -18085.368} C_VEL
LIN {X 0,Y 261.117,Z 626.366,A -85,B 0,C 180,E1 -18088.458,E2 -18088.458} C_VEL
LIN {X 0,Y 261.111,Z 626.928,A -85,B 0,C 180,E1 -18091.542,E2 -18091.542} C_VEL
LIN {X 0,Y 261.045,Z 626.151,A -85,B 0,C 180,E1 -18094.633,E2 -18094.633} C_VEL
LIN {X 0,Y 261.289,Z 624.035,A -85,B 0,C 180,E1 -18097.729,E2 -18097.729} C_VEL
LIN {X 0,Y 261.94,Z 620.533,A -85,B 0,C 180,E1 -18100.825,E2 -18100.825} C_VEL
LIN {X 0,Y 263.195,Z 615.547,A -85,B 0,C 180,E1 -18103.906,E2 -18103.906} C_VEL
LIN {X 0,Y 265.057,Z 608.935,A -85,B 0,C 180,E1 -18106.958,E2 -18106.958} C_VEL
LIN {X 0,Y 267.141,Z 601.598,A -85,B 0,C 180,E1 -18109.599,E2 -18109.599} C_VEL
LIN {X 0,Y 269.903,Z 592.51,A -85,B 0,C 180,E1 -18112.183,E2 -18112.183} C_VEL
LIN {X 0,Y 272.71,Z 583.017,A -85,B 0,C 180,E1 -18114.352,E2 -18114.352} C_VEL
LIN {X 0,Y 275.664,Z 572.518,A -85,B 0,C 180,E1 -18116.294,E2 -18116.294} C_VEL
LIN {X 0,Y 278.472,Z 561.064,A -85,B 0,C 180,E1 -18118.019,E2 -18118.019} C_VEL
LIN {X 0,Y 281.318,Z 548.112,A -85,B 0,C 180,E1 -18119.565,E2 -18119.565} C_VEL
LIN {X 0,Y 283.705,Z 535.563,A -85,B 0,C 180,E1 -18120.726,E2 -18120.726} C_VEL
LIN {X 0,Y 285.925,Z 521.582,A -85,B 0,C 180,E1 -18121.695,E2 -18121.695} C_VEL
LIN {X 0,Y 287.535,Z 507.731,A -85,B 0,C 180,E1 -18122.374,E2 -18122.374} C_VEL
LIN {X 0,Y 288.424,Z 493.903,A -85,B 0,C 180,E1 -18122.817,E2 -18122.817} C_VEL
LIN {X 0,Y 291.431,Z 419.307,A -85,B 0,C 180,E1 -18124.62,E2 -18124.62} C_VEL
LIN {X 0,Y 289.439,Z 407.917,A -85,B 0,C 180,E1 -18125.261,E2 -18125.261} C_VEL
LIN {X 0,Y 282.635,Z 392.587,A -85,B 0,C 180,E1 -18126.805,E2 -18126.805} C_VEL
LIN {X 0,Y 275.79,Z 379.208,A -85,B 0,C 180,E1 -18128.405,E2 -18128.405} C_VEL
LIN {X 0,Y 270.657,Z 369.98,A -85,B 0,C 180,E1 -18129.657,E2 -18129.657} C_VEL
LIN {X 0,Y 266.455,Z 362.467,A -85,B 0,C 180,E1 -18130.755,E2 -18130.755} C_VEL
LIN {X 0,Y 263.858,Z 353.862,A -85,B 0,C 180,E1 -18134.562,E2 -18134.562} C_VEL
LIN {X 0,Y 263.103,Z 351.331,A -85,B 0,C 180,E1 -18135.746,E2 -18135.746} C_VEL
LIN {X 0,Y 263.125,Z 351.328,A -85,B 0,C 180,E1 -18138.407,E2 -18138.407} C_VEL
LIN {X 0,Y 263.167,Z 351.328,A -85,B 0,C 180,E1 -18142.105,E2 -18142.105} C_VEL
LIN {X 0,Y 263.185,Z 351.324,A -85,B 0,C 180,E1 -18145.891,E2 -18145.891} C_VEL
LIN {X 0,Y 263.127,Z 351.329,A -85,B 0,C 180,E1 -18149.504,E2 -18149.504} C_VEL
LIN {X 0,Y 263.146,Z 351.326,A -85,B 0,C 180,E1 -18152.998,E2 -18152.998} C_VEL
LIN {X 0,Y 263.151,Z 351.329,A -85,B 0,C 180,E1 -18156.384,E2 -18156.384} C_VEL
LIN {X 0,Y 263.265,Z 351.316,A -85,B 0,C 180,E1 -18159.694,E2 -18159.694} C_VEL
LIN {X 0,Y 263.354,Z 351.306,A -85,B 0,C 180,E1 -18164.523,E2 -18164.523} C_VEL
LIN {X 0,Y 263.357,Z 351.305,A -85,B 0,C 180,E1 -18169.234,E2 -18169.234} C_VEL
LIN {X 0,Y 263.529,Z 351.272,A -85,B 0,C 180,E1 -18172.338,E2 -18172.338} C_VEL
LIN {X 0,Y 263.742,Z 351.255,A -85,B 0,C 180,E1 -18178.473,E2 -18178.473} C_VEL
LIN {X 0,Y 263.744,Z 351.244,A -85,B 0,C 180,E1 -18181.527,E2 -18181.527} C_VEL
LIN {X 0,Y 263.529,Z 351.271,A -85,B 0,C 180,E1 -18187.663,E2 -18187.663} C_VEL
LIN {X 0,Y 263.347,Z 351.299,A -85,B 0,C 180,E1 -18190.767,E2 -18190.767} C_VEL
LIN {X 0,Y 263.291,Z 351.305,A -85,B 0,C 180,E1 -18195.482,E2 -18195.482} C_VEL
LIN {X 0,Y 263.21,Z 351.313,A -85,B 0,C 180,E1 -18200.312,E2 -18200.312} C_VEL
LIN {X 0,Y 263.107,Z 351.327,A -85,B 0,C 180,E1 -18205.302,E2 -18205.302} C_VEL
LIN {X 0,Y 263.12,Z 351.311,A -85,B 0,C 180,E1 -18208.737,E2 -18208.737} C_VEL
LIN {X 0,Y 263.129,Z 351.316,A -85,B 0,C 180,E1 -18212.289,E2 -18212.289} C_VEL
LIN {X 0,Y 263.178,Z 351.3,A -85,B 0,C 180,E1 -18216.761,E2 -18216.761} C_VEL
LIN {X 0,Y 263.094,Z 351.335,A -85,B 0,C 180,E1 -18219.875,E2 -18219.875} C_VEL
LIN {X 0,Y 263.109,Z 351.36,A -85,B 0,C 180,E1 -18223.417,E2 -18223.417} C_VEL
LIN {X 0,Y 263.173,Z 351.897,A -85,B 0,C 180,E1 -18223.647,E2 -18223.647} C_VEL
LIN {X 0,Y 264.361,Z 354.589,A -85,B 0,C 180,E1 -18223.992,E2 -18223.992} C_VEL
LIN {X 0,Y 266.242,Z 356.823,A -85,B 0,C 180,E1 -18224.456,E2 -18224.456} C_VEL
LIN {X 0,Y 272.334,Z 366.532,A -85,B 0,C 180,E1 -18225.976,E2 -18225.976} C_VEL
LIN {X 0,Y 280.701,Z 381.227,A -85,B 0,C 180,E1 -18227.947,E2 -18227.947} C_VEL
LIN {X 0,Y 287.927,Z 395.85,A -85,B 0,C 180,E1 -18229.576,E2 -18229.576} C_VEL
LIN {X 0,Y 291.988,Z 405.113,A -85,B 0,C 180,E1 -18230.472,E2 -18230.472} C_VEL
LIN {X 0,Y 288.586,Z 487.548,A -85,B 0,C 180,E1 -18232.495,E2 -18232.495} C_VEL
LIN {X 0,Y 287.332,Z 502.36,A -85,B 0,C 180,E1 -18233.128,E2 -18233.128} C_VEL
LIN {X 0,Y 285.457,Z 516.362,A -85,B 0,C 180,E1 -18233.993,E2 -18233.993} C_VEL
LIN {X 0,Y 283.369,Z 528.4,A -85,B 0,C 180,E1 -18234.983,E2 -18234.983} C_VEL
LIN {X 0,Y 280.951,Z 541.367,A -85,B 0,C 180,E1 -18236.395,E2 -18236.395} C_VEL
LIN {X 0,Y 278.152,Z 552.973,A -85,B 0,C 180,E1 -18237.954,E2 -18237.954} C_VEL
LIN {X 0,Y 275.438,Z 563.6,A -85,B 0,C 180,E1 -18239.739,E2 -18239.739} C_VEL
LIN {X 0,Y 272.631,Z 574.119,A -85,B 0,C 180,E1 -18241.936,E2 -18241.936} C_VEL
LIN {X 0,Y 269.954,Z 582.767,A -85,B 0,C 180,E1 -18244.146,E2 -18244.146} C_VEL
LIN {X 0,Y 267.363,Z 591.019,A -85,B 0,C 180,E1 -18246.778,E2 -18246.778} C_VEL
LIN {X 0,Y 265.59,Z 596.769,A -85,B 0,C 180,E1 -18249.069,E2 -18249.069} C_VEL
LIN {X 0,Y 264.112,Z 601.46,A -85,B 0,C 180,E1 -18251.378,E2 -18251.378} C_VEL
LIN {X 0,Y 262.676,Z 606.301,A -85,B 0,C 180,E1 -18254.481,E2 -18254.481} C_VEL
LIN {X 0,Y 261.668,Z 609.635,A -85,B 0,C 180,E1 -18257.592,E2 -18257.592} C_VEL
LIN {X 0,Y 261.184,Z 611.558,A -85,B 0,C 180,E1 -18260.709,E2 -18260.709} C_VEL
LIN {X 0,Y 261.127,Z 612.13,A -85,B 0,C 180,E1 -18263.82,E2 -18263.82} C_VEL
LIN {X 0,Y 261.111,Z 611.387,A -85,B 0,C 180,E1 -18266.914,E2 -18266.914} C_VEL
LIN {X 0,Y 261.204,Z 609.327,A -85,B 0,C 180,E1 -18270,E2 -18270} C_VEL
LIN {X 0,Y 261.625,Z 605.896,A -85,B 0,C 180,E1 -18273.08,E2 -18273.08} C_VEL
LIN {X 0,Y 262.581,Z 600.987,A -85,B 0,C 180,E1 -18276.146,E2 -18276.146} C_VEL
LIN {X 0,Y 264.02,Z 594.451,A -85,B 0,C 180,E1 -18279.19,E2 -18279.19} C_VEL
LIN {X 0,Y 265.514,Z 587.25,A -85,B 0,C 180,E1 -18281.818,E2 -18281.818} C_VEL
LIN {X 0,Y 267.128,Z 579.589,A -85,B 0,C 180,E1 -18284.085,E2 -18284.085} C_VEL
LIN {X 0,Y 269.412,Z 570.443,A -85,B 0,C 180,E1 -18286.286,E2 -18286.286} C_VEL
LIN {X 0,Y 271.512,Z 560.37,A -85,B 0,C 180,E1 -18288.292,E2 -18288.292} C_VEL
LIN {X 0,Y 273.628,Z 549.3,A -85,B 0,C 180,E1 -18290.092,E2 -18290.092} C_VEL
LIN {X 0,Y 275.838,Z 537.06,A -85,B 0,C 180,E1 -18291.681,E2 -18291.681} C_VEL
LIN {X 0,Y 277.856,Z 523.35,A -85,B 0,C 180,E1 -18293.082,E2 -18293.082} C_VEL
LIN {X 0,Y 279.536,Z 509.935,A -85,B 0,C 180,E1 -18294.114,E2 -18294.114} C_VEL
LIN {X 0,Y 280.79,Z 496.119,A -85,B 0,C 180,E1 -18294.886,E2 -18294.886} C_VEL
LIN {X 0,Y 281.616,Z 482.186,A -85,B 0,C 180,E1 -18295.388,E2 -18295.388} C_VEL
LIN {X 0,Y 284.551,Z 397.695,A -85,B 0,C 180,E1 -18297.475,E2 -18297.475} C_VEL
LIN {X 0,Y 277.825,Z 381.05,A -85,B 0,C 180,E1 -18298.79,E2 -18298.79} C_VEL
LIN {X 0,Y 269.193,Z 362.755,A -85,B 0,C 180,E1 -18300.507,E2 -18300.507} C_VEL
LIN {X 0,Y 266.438,Z 357.954,A -85,B 0,C 180,E1 -18301.053,E2 -18301.053} C_VEL
LIN {X 0,Y 264.559,Z 354.785,A -85,B 0,C 180,E1 -18301.43,E2 -18301.43} C_VEL
LIN {X 0,Y 263.299,Z 352.287,A -85,B 0,C 180,E1 -18301.699,E2 -18301.699} C_VEL
LIN {X 0,Y 263.128,Z 351.336,A -85,B 0,C 180,E1 -18301.794,E2 -18301.794} C_VEL
LIN {X 0,Y 263.159,Z 351.33,A -85,B 0,C 180,E1 -18305.983,E2 -18305.983} C_VEL
LIN {X 0,Y 263.094,Z 351.336,A -85,B 0,C 180,E1 -18309.875,E2 -18309.875} C_VEL
LIN {X 0,Y 263.079,Z 351.34,A -85,B 0,C 180,E1 -18313.994,E2 -18313.994} C_VEL
LIN {X 0,Y 263.082,Z 351.333,A -85,B 0,C 180,E1 -18318.417,E2 -18318.417} C_VEL
LIN {X 0,Y 263.117,Z 351.329,A -85,B 0,C 180,E1 -18322.095,E2 -18322.095} C_VEL
LIN {X 0,Y 263.154,Z 351.329,A -85,B 0,C 180,E1 -18325.885,E2 -18325.885} C_VEL
LIN {X 0,Y 263.111,Z 351.335,A -85,B 0,C 180,E1 -18329.501,E2 -18329.501} C_VEL
LIN {X 0,Y 263.096,Z 351.326,A -85,B 0,C 180,E1 -18333.436,E2 -18333.436} C_VEL
LIN {X 0,Y 263.127,Z 351.33,A -85,B 0,C 180,E1 -18336.381,E2 -18336.381} C_VEL
LIN {X 0,Y 263.18,Z 351.293,A -85,B 0,C 180,E1 -18340.074,E2 -18340.074} C_VEL
LIN {X 0,Y 262.463,Z 351.395,A -85,B 0,C 180,E1 -18341.351,E2 -18341.351} C_VEL
LIN {X 0,Y 259.612,Z 351.769,A -85,B 0,C 180,E1 -18343.435,E2 -18343.435} C_VEL
LIN {X 0,Y 257.25,Z 352.063,A -85,B 0,C 180,E1 -18345.13,E2 -18345.13} C_VEL
LIN {X 0,Y 256.278,Z 352.173,A -85,B 0,C 180,E1 -18346.444,E2 -18346.444} C_VEL
LIN {X 0,Y 256.218,Z 352.171,A -85,B 0,C 180,E1 -18346.888,E2 -18346.888} C_VEL
LIN {X 0,Y 256.415,Z 352.141,A -85,B 0,C 180,E1 -18350.651,E2 -18350.651} C_VEL
LIN {X 0,Y 256.46,Z 352.164,A -85,B 0,C 180,E1 -18353.706,E2 -18353.706} C_VEL
LIN {X 0,Y 256.707,Z 352.135,A -85,B 0,C 180,E1 -18358.431,E2 -18358.431} C_VEL
LIN {X 0,Y 256.703,Z 352.125,A -85,B 0,C 180,E1 -18361.568,E2 -18361.568} C_VEL
LIN {X 0,Y 256.458,Z 352.159,A -85,B 0,C 180,E1 -18366.293,E2 -18366.293} C_VEL
LIN {X 0,Y 256.429,Z 352.164,A -85,B 0,C 180,E1 -18369.464,E2 -18369.464} C_VEL
LIN {X 0,Y 256.257,Z 352.183,A -85,B 0,C 180,E1 -18374.29,E2 -18374.29} C_VEL
LIN {X 0,Y 256.213,Z 352.192,A -85,B 0,C 180,E1 -18377.561,E2 -18377.561} C_VEL
LIN {X 0,Y 256.157,Z 352.201,A -85,B 0,C 180,E1 -18381.118,E2 -18381.118} C_VEL
LIN {X 0,Y 256.168,Z 352.199,A -85,B 0,C 180,E1 -18385.128,E2 -18385.128} C_VEL
LIN {X 0,Y 256.113,Z 352.206,A -85,B 0,C 180,E1 -18388.584,E2 -18388.584} C_VEL
LIN {X 0,Y 256.084,Z 352.211,A -85,B 0,C 180,E1 -18393.29,E2 -18393.29} C_VEL
LIN {X 0,Y 256.13,Z 352.211,A -85,B 0,C 180,E1 -18397.275,E2 -18397.275} C_VEL
LIN {X 0,Y 256.057,Z 352.219,A -85,B 0,C 180,E1 -18401.202,E2 -18401.202} C_VEL
LIN {X 0,Y 256.058,Z 352.216,A -85,B 0,C 180,E1 -18405.53,E2 -18405.53} C_VEL
LIN {X 0,Y 256.111,Z 352.328,A -85,B 0,C 180,E1 -18408.468,E2 -18408.468} C_VEL
LIN {X 0,Y 258.551,Z 361.308,A -85,B 0,C 180,E1 -18412.025,E2 -18412.025} C_VEL
LIN {X 0,Y 259.015,Z 363.187,A -85,B 0,C 180,E1 -18412.644,E2 -18412.644} C_VEL
LIN {X 0,Y 265.884,Z 377.381,A -85,B 0,C 180,E1 -18414.124,E2 -18414.124} C_VEL
LIN {X 0,Y 273.668,Z 395.359,A -85,B 0,C 180,E1 -18415.743,E2 -18415.743} C_VEL
LIN {X 0,Y 275.494,Z 400.923,A -85,B 0,C 180,E1 -18416.145,E2 -18416.145} C_VEL
LIN {X 0,Y 277.82,Z 418.163,A -85,B 0,C 180,E1 -18416.948,E2 -18416.948} C_VEL
LIN {X 0,Y 274.777,Z 501.397,A -85,B 0,C 180,E1 -18419.073,E2 -18419.073} C_VEL
LIN {X 0,Y 273.487,Z 516.058,A -85,B 0,C 180,E1 -18419.714,E2 -18419.714} C_VEL
LIN {X 0,Y 271.914,Z 529.505,A -85,B 0,C 180,E1 -18420.588,E2 -18420.588} C_VEL
LIN {X 0,Y 270.053,Z 541.758,A -85,B 0,C 180,E1 -18421.644,E2 -18421.644} C_VEL
LIN {X 0,Y 267.897,Z 554.225,A -85,B 0,C 180,E1 -18423.031,E2 -18423.031} C_VEL
LIN {X 0,Y 265.483,Z 566.373,A -85,B 0,C 180,E1 -18424.732,E2 -18424.732} C_VEL
LIN {X 0,Y 263.356,Z 576.104,A -85,B 0,C 180,E1 -18426.403,E2 -18426.403} C_VEL
LIN {X 0,Y 260.872,Z 586.896,A -85,B 0,C 180,E1 -18428.673,E2 -18428.673} C_VEL
LIN {X 0,Y 258.796,Z 595.801,A -85,B 0,C 180,E1 -18430.981,E2 -18430.981} C_VEL
LIN {X 0,Y 257.304,Z 603.449,A -85,B 0,C 180,E1 -18433.417,E2 -18433.417} C_VEL
LIN {X 0,Y 256.049,Z 609.38,A -85,B 0,C 180,E1 -18435.698,E2 -18435.698} C_VEL
LIN {X 0,Y 255.012,Z 614.481,A -85,B 0,C 180,E1 -18438.071,E2 -18438.071} C_VEL
LIN {X 0,Y 254.323,Z 619.734,A -85,B 0,C 180,E1 -18441.258,E2 -18441.258} C_VEL
LIN {X 0,Y 254.053,Z 622.68,A -85,B 0,C 180,E1 -18443.647,E2 -18443.647} C_VEL
LIN {X 0,Y 253.981,Z 625.338,A -85,B 0,C 180,E1 -18446.828,E2 -18446.828} C_VEL
LIN {X 0,Y 254.054,Z 626.608,A -85,B 0,C 180,E1 -18450,E2 -18450} C_VEL
LIN {X 0,Y 254.016,Z 626.733,A -85,B 0,C 180,E1 -18451.586,E2 -18451.586} C_VEL
LIN {X 0,Y 253.972,Z 625.979,A -85,B 0,C 180,E1 -18454.762,E2 -18454.762} C_VEL
LIN {X 0,Y 254.229,Z 623.887,A -85,B 0,C 180,E1 -18457.945,E2 -18457.945} C_VEL
LIN {X 0,Y 254.936,Z 620.41,A -85,B 0,C 180,E1 -18461.127,E2 -18461.127} C_VEL
LIN {X 0,Y 256.273,Z 615.451,A -85,B 0,C 180,E1 -18464.289,E2 -18464.289} C_VEL
LIN {X 0,Y 258.194,Z 608.868,A -85,B 0,C 180,E1 -18467.423,E2 -18467.423} C_VEL
LIN {X 0,Y 260.434,Z 601.565,A -85,B 0,C 180,E1 -18470.125,E2 -18470.125} C_VEL
LIN {X 0,Y 263.318,Z 592.534,A -85,B 0,C 180,E1 -18472.769,E2 -18472.769} C_VEL
LIN {X 0,Y 266.25,Z 583.085,A -85,B 0,C 180,E1 -18474.983,E2 -18474.983} C_VEL
LIN {X 0,Y 269.328,Z 572.64,A -85,B 0,C 180,E1 -18476.962,E2 -18476.962} C_VEL
LIN {X 0,Y 272.145,Z 561.582,A -85,B 0,C 180,E1 -18478.677,E2 -18478.677} C_VEL
LIN {X 0,Y 274.837,Z 549.967,A -85,B 0,C 180,E1 -18480.122,E2 -18480.122} C_VEL
LIN {X 0,Y 277.299,Z 537.945,A -85,B 0,C 180,E1 -18481.303,E2 -18481.303} C_VEL
LIN {X 0,Y 279.568,Z 524.757,A -85,B 0,C 180,E1 -18482.29,E2 -18482.29} C_VEL
LIN {X 0,Y 281.381,Z 510.475,A -85,B 0,C 180,E1 -18483.065,E2 -18483.065} C_VEL
LIN {X 0,Y 282.469,Z 496.91,A -85,B 0,C 180,E1 -18483.552,E2 -18483.552} C_VEL
LIN {X 0,Y 285.73,Z 420.549,A -85,B 0,C 180,E1 -18485.435,E2 -18485.435} C_VEL
LIN {X 0,Y 283.992,Z 410.644,A -85,B 0,C 180,E1 -18486.015,E2 -18486.015} C_VEL
LIN {X 0,Y 277.318,Z 395.601,A -85,B 0,C 180,E1 -18487.594,E2 -18487.594} C_VEL
LIN {X 0,Y 269.901,Z 381.019,A -85,B 0,C 180,E1 -18489.415,E2 -18489.415} C_VEL
LIN {X 0,Y 263.516,Z 369.85,A -85,B 0,C 180,E1 -18491.06,E2 -18491.06} C_VEL
LIN {X 0,Y 261.448,Z 366.344,A -85,B 0,C 180,E1 -18491.615,E2 -18491.615} C_VEL
LIN {X 0,Y 259.038,Z 362.127,A -85,B 0,C 180,E1 -18492.328,E2 -18492.328} C_VEL
LIN {X 0,Y 256.814,Z 354.661,A -85,B 0,C 180,E1 -18495.81,E2 -18495.81} C_VEL
LIN {X 0,Y 256.051,Z 352.214,A -85,B 0,C 180,E1 -18497.073,E2 -18497.073} C_VEL
LIN {X 0,Y 256.089,Z 352.203,A -85,B 0,C 180,E1 -18500.862,E2 -18500.862} C_VEL
LIN {X 0,Y 256.122,Z 352.205,A -85,B 0,C 180,E1 -18504.814,E2 -18504.814} C_VEL
LIN {X 0,Y 256.084,Z 352.212,A -85,B 0,C 180,E1 -18508.572,E2 -18508.572} C_VEL
LIN {X 0,Y 256.098,Z 352.21,A -85,B 0,C 180,E1 -18512.191,E2 -18512.191} C_VEL
LIN {X 0,Y 256.137,Z 352.204,A -85,B 0,C 180,E1 -18515.696,E2 -18515.696} C_VEL
LIN {X 0,Y 256.165,Z 352.197,A -85,B 0,C 180,E1 -18519.105,E2 -18519.105} C_VEL
LIN {X 0,Y 256.303,Z 352.183,A -85,B 0,C 180,E1 -18524.086,E2 -18524.086} C_VEL
LIN {X 0,Y 256.297,Z 352.171,A -85,B 0,C 180,E1 -18527.328,E2 -18527.328} C_VEL
LIN {X 0,Y 256.437,Z 352.16,A -85,B 0,C 180,E1 -18530.623,E2 -18530.623} C_VEL
LIN {X 0,Y 256.459,Z 352.163,A -85,B 0,C 180,E1 -18533.707,E2 -18533.707} C_VEL
LIN {X 0,Y 256.704,Z 352.131,A -85,B 0,C 180,E1 -18538.432,E2 -18538.432} C_VEL
LIN {X 0,Y 256.707,Z 352.12,A -85,B 0,C 180,E1 -18541.569,E2 -18541.569} C_VEL
LIN {X 0,Y 256.448,Z 352.15,A -85,B 0,C 180,E1 -18546.564,E2 -18546.564} C_VEL
LIN {X 0,Y 256.43,Z 352.17,A -85,B 0,C 180,E1 -18549.465,E2 -18549.465} C_VEL
LIN {X 0,Y 256.211,Z 352.195,A -85,B 0,C 180,E1 -18554.293,E2 -18554.293} C_VEL
LIN {X 0,Y 256.15,Z 352.196,A -85,B 0,C 180,E1 -18557.567,E2 -18557.567} C_VEL
LIN {X 0,Y 256.121,Z 352.195,A -85,B 0,C 180,E1 -18561.097,E2 -18561.097} C_VEL
LIN {X 0,Y 256.08,Z 352.202,A -85,B 0,C 180,E1 -18565.085,E2 -18565.085} C_VEL
LIN {X 0,Y 256.078,Z 352.189,A -85,B 0,C 180,E1 -18568.569,E2 -18568.569} C_VEL
LIN {X 0,Y 256.072,Z 352.184,A -85,B 0,C 180,E1 -18571.7,E2 -18571.7} C_VEL
LIN {X 0,Y 256.082,Z 352.192,A -85,B 0,C 180,E1 -18575.194,E2 -18575.194} C_VEL
LIN {X 0,Y 256.068,Z 352.215,A -85,B 0,C 180,E1 -18579.143,E2 -18579.143} C_VEL
LIN {X 0,Y 256.063,Z 352.213,A -85,B 0,C 180,E1 -18582.099,E2 -18582.099} C_VEL
LIN {X 0,Y 256.987,Z 354.933,A -85,B 0,C 180,E1 -18582.425,E2 -18582.425} C_VEL
LIN {X 0,Y 259.22,Z 357.573,A -85,B 0,C 180,E1 -18583.018,E2 -18583.018} C_VEL
LIN {X 0,Y 261.198,Z 360.724,A -85,B 0,C 180,E1 -18583.561,E2 -18583.561} C_VEL
LIN {X 0,Y 262.659,Z 362.775,A -85,B 0,C 180,E1 -18583.942,E2 -18583.942} C_VEL
LIN {X 0,Y 265.773,Z 367.607,A -85,B 0,C 180,E1 -18584.751,E2 -18584.751} C_VEL
LIN {X 0,Y 272.737,Z 379.485,A -85,B 0,C 180,E1 -18586.495,E2 -18586.495} C_VEL
LIN {X 0,Y 279.707,Z 392.8,A -85,B 0,C 180,E1 -18588.156,E2 -18588.156} C_VEL
LIN {X 0,Y 285.502,Z 405.481,A -85,B 0,C 180,E1 -18589.498,E2 -18589.498} C_VEL
LIN {X 0,Y 286.242,Z 407.178,A -85,B 0,C 180,E1 -18589.667,E2 -18589.667} C_VEL
LIN {X 0,Y 282.758,Z 488.25,A -85,B 0,C 180,E1 -18591.696,E2 -18591.696} C_VEL
LIN {X 0,Y 281.455,Z 502.886,A -85,B 0,C 180,E1 -18592.338,E2 -18592.338} C_VEL
LIN {X 0,Y 279.446,Z 517.195,A -85,B 0,C 180,E1 -18593.244,E2 -18593.244} C_VEL
LIN {X 0,Y 277.018,Z 530.895,A -85,B 0,C 180,E1 -18594.433,E2 -18594.433} C_VEL
LIN {X 0,Y 274.351,Z 543.872,A -85,B 0,C 180,E1 -18595.918,E2 -18595.918} C_VEL
LIN {X 0,Y 271.485,Z 555.066,A -85,B 0,C 180,E1 -18597.509,E2 -18597.509} C_VEL
LIN {X 0,Y 268.72,Z 565.374,A -85,B 0,C 180,E1 -18599.337,E2 -18599.337} C_VEL
LIN {X 0,Y 265.803,Z 575.571,A -85,B 0,C 180,E1 -18601.58,E2 -18601.58} C_VEL
LIN {X 0,Y 263.049,Z 584.003,A -85,B 0,C 180,E1 -18603.842,E2 -18603.842} C_VEL
LIN {X 0,Y 260.746,Z 591.018,A -85,B 0,C 180,E1 -18606.152,E2 -18606.152} C_VEL
LIN {X 0,Y 258.876,Z 596.792,A -85,B 0,C 180,E1 -18608.5,E2 -18608.5} C_VEL
LIN {X 0,Y 257.276,Z 601.521,A -85,B 0,C 180,E1 -18610.864,E2 -18610.864} C_VEL
LIN {X 0,Y 255.702,Z 606.535,A -85,B 0,C 180,E1 -18614.153,E2 -18614.153} C_VEL
LIN {X 0,Y 254.65,Z 609.765,A -85,B 0,C 180,E1 -18617.244,E2 -18617.244} C_VEL
LIN {X 0,Y 254.124,Z 611.728,A -85,B 0,C 180,E1 -18620.448,E2 -18620.448} C_VEL
LIN {X 0,Y 254.028,Z 612.339,A -85,B 0,C 180,E1 -18623.646,E2 -18623.646} C_VEL
LIN {X 0,Y 254.005,Z 611.629,A -85,B 0,C 180,E1 -18626.828,E2 -18626.828} C_VEL
LIN {X 0,Y 254.085,Z 610.779,A -85,B 0,C 180,E1 -18628.415,E2 -18628.415} C_VEL
LIN {X 0,Y 254.29,Z 608.077,A -85,B 0,C 180,E1 -18631.584,E2 -18631.584} C_VEL
LIN {X 0,Y 254.982,Z 603.959,A -85,B 0,C 180,E1 -18634.743,E2 -18634.743} C_VEL
LIN {X 0,Y 256.254,Z 598.293,A -85,B 0,C 180,E1 -18637.882,E2 -18637.882} C_VEL
LIN {X 0,Y 257.548,Z 592.906,A -85,B 0,C 180,E1 -18640.217,E2 -18640.217} C_VEL
LIN {X 0,Y 259.063,Z 585.228,A -85,B 0,C 180,E1 -18642.933,E2 -18642.933} C_VEL
LIN {X 0,Y 261.03,Z 577.195,A -85,B 0,C 180,E1 -18645.219,E2 -18645.219} C_VEL
LIN {X 0,Y 263.398,Z 567.511,A -85,B 0,C 180,E1 -18647.468,E2 -18647.468} C_VEL
LIN {X 0,Y 265.633,Z 556.786,A -85,B 0,C 180,E1 -18649.513,E2 -18649.513} C_VEL
LIN {X 0,Y 267.962,Z 544.893,A -85,B 0,C 180,E1 -18651.34,E2 -18651.34} C_VEL
LIN {X 0,Y 270.082,Z 533.173,A -85,B 0,C 180,E1 -18652.773,E2 -18652.773} C_VEL
LIN {X 0,Y 271.986,Z 520.379,A -85,B 0,C 180,E1 -18654.015,E2 -18654.015} C_VEL
LIN {X 0,Y 273.569,Z 507.267,A -85,B 0,C 180,E1 -18654.979,E2 -18654.979} C_VEL
LIN {X 0,Y 274.75,Z 493.029,A -85,B 0,C 180,E1 -18655.725,E2 -18655.725} C_VEL
LIN {X 0,Y 275.515,Z 477.816,A -85,B 0,C 180,E1 -18656.213,E2 -18656.213} C_VEL
LIN {X 0,Y 278.402,Z 399.418,A -85,B 0,C 180,E1 -18658.172,E2 -18658.172} C_VEL
LIN {X 0,Y 271.402,Z 382.262,A -85,B 0,C 180,E1 -18659.597,E2 -18659.597} C_VEL
LIN {X 0,Y 263.977,Z 366.635,A -85,B 0,C 180,E1 -18661.134,E2 -18661.134} C_VEL
LIN {X 0,Y 259.718,Z 359.291,A -85,B 0,C 180,E1 -18662.015,E2 -18662.015} C_VEL
LIN {X 0,Y 257.6,Z 355.798,A -85,B 0,C 180,E1 -18662.462,E2 -18662.462} C_VEL
LIN {X 0,Y 256.297,Z 353.312,A -85,B 0,C 180,E1 -18662.754,E2 -18662.754} C_VEL
LIN {X 0,Y 256.085,Z 352.209,A -85,B 0,C 180,E1 -18662.88,E2 -18662.88} C_VEL
LIN {X 0,Y 256.118,Z 352.205,A -85,B 0,C 180,E1 -18667.271,E2 -18667.271} C_VEL
LIN {X 0,Y 256.021,Z 352.217,A -85,B 0,C 180,E1 -18671.21,E2 -18671.21} C_VEL
LIN {X 0,Y 256.02,Z 352.214,A -85,B 0,C 180,E1 -18675.539,E2 -18675.539} C_VEL
LIN {X 0,Y 256.018,Z 352.212,A -85,B 0,C 180,E1 -18678.789,E2 -18678.789} C_VEL
LIN {X 0,Y 256.101,Z 352.2,A -85,B 0,C 180,E1 -18682.862,E2 -18682.862} C_VEL
LIN {X 0,Y 256.068,Z 352.203,A -85,B 0,C 180,E1 -18686.707,E2 -18686.707} C_VEL
LIN {X 0,Y 256.043,Z 352.216,A -85,B 0,C 180,E1 -18690.391,E2 -18690.391} C_VEL
LIN {X 0,Y 256.07,Z 352.206,A -85,B 0,C 180,E1 -18693.951,E2 -18693.951} C_VEL
LIN {X 0,Y 256.065,Z 352.201,A -85,B 0,C 180,E1 -18697.402,E2 -18697.402} C_VEL
LIN {X 0,Y 256.11,Z 352.177,A -85,B 0,C 180,E1 -18700.773,E2 -18700.773} C_VEL
LIN {X 0,Y 256.216,Z 352.195,A -85,B 0,C 180,E1 -18704.079,E2 -18704.079} C_VEL
LIN {X 0,Y 256.218,Z 352.171,A -85,B 0,C 180,E1 -18706.888,E2 -18706.888} C_VEL
LIN {X 0,Y 255.646,Z 352.237,A -85,B 0,C 180,E1 -18708.202,E2 -18708.202} C_VEL
LIN {X 0,Y 252.972,Z 352.583,A -85,B 0,C 180,E1 -18710.348,E2 -18710.348} C_VEL
LIN {X 0,Y 249.774,Z 352.996,A -85,B 0,C 180,E1 -18712.989,E2 -18712.989} C_VEL
LIN {X 0,Y 249.379,Z 353.042,A -85,B 0,C 180,E1 -18713.901,E2 -18713.901} C_VEL
LIN {X 0,Y 249.669,Z 353.012,A -85,B 0,C 180,E1 -18718.386,E2 -18718.386} C_VEL
LIN {X 0,Y 249.664,Z 353.002,A -85,B 0,C 180,E1 -18721.613,E2 -18721.613} C_VEL
LIN {X 0,Y 249.432,Z 353.035,A -85,B 0,C 180,E1 -18726.471,E2 -18726.471} C_VEL
LIN {X 0,Y 249.345,Z 353.044,A -85,B 0,C 180,E1 -18729.736,E2 -18729.736} C_VEL
LIN {X 0,Y 249.208,Z 353.062,A -85,B 0,C 180,E1 -18734.703,E2 -18734.703} C_VEL
LIN {X 0,Y 249.142,Z 353.07,A -85,B 0,C 180,E1 -18738.077,E2 -18738.077} C_VEL
LIN {X 0,Y 249.086,Z 353.079,A -85,B 0,C 180,E1 -18741.518,E2 -18741.518} C_VEL
LIN {X 0,Y 249.114,Z 353.076,A -85,B 0,C 180,E1 -18745.473,E2 -18745.473} C_VEL
LIN {X 0,Y 249.055,Z 353.084,A -85,B 0,C 180,E1 -18748.981,E2 -18748.981} C_VEL
LIN {X 0,Y 249.034,Z 353.087,A -85,B 0,C 180,E1 -18752.425,E2 -18752.425} C_VEL
LIN {X 0,Y 249.07,Z 353.087,A -85,B 0,C 180,E1 -18756.338,E2 -18756.338} C_VEL
LIN {X 0,Y 249.027,Z 353.093,A -85,B 0,C 180,E1 -18760.474,E2 -18760.474} C_VEL
LIN {X 0,Y 249.003,Z 353.095,A -85,B 0,C 180,E1 -18764.879,E2 -18764.879} C_VEL
LIN {X 0,Y 249.032,Z 353.138,A -85,B 0,C 180,E1 -18767.521,E2 -18767.521} C_VEL
LIN {X 0,Y 251.638,Z 362.702,A -85,B 0,C 180,E1 -18771.445,E2 -18771.445} C_VEL
LIN {X 0,Y 259.967,Z 379.649,A -85,B 0,C 180,E1 -18773.332,E2 -18773.332} C_VEL
LIN {X 0,Y 267.758,Z 397.65,A -85,B 0,C 180,E1 -18775.024,E2 -18775.024} C_VEL
LIN {X 0,Y 269.573,Z 402.883,A -85,B 0,C 180,E1 -18775.432,E2 -18775.432} C_VEL
LIN {X 0,Y 271.73,Z 419.079,A -85,B 0,C 180,E1 -18776.211,E2 -18776.211} C_VEL
LIN {X 0,Y 268.6,Z 501.019,A -85,B 0,C 180,E1 -18778.339,E2 -18778.339} C_VEL
LIN {X 0,Y 267.393,Z 514.932,A -85,B 0,C 180,E1 -18778.948,E2 -18778.948} C_VEL
LIN {X 0,Y 265.911,Z 527.478,A -85,B 0,C 180,E1 -18779.747,E2 -18779.747} C_VEL
LIN {X 0,Y 263.772,Z 541.014,A -85,B 0,C 180,E1 -18780.905,E2 -18780.905} C_VEL
LIN {X 0,Y 261.686,Z 552.574,A -85,B 0,C 180,E1 -18782.185,E2 -18782.185} C_VEL
LIN {X 0,Y 259.242,Z 564.878,A -85,B 0,C 180,E1 -18783.909,E2 -18783.909} C_VEL
LIN {X 0,Y 256.791,Z 575.6,A -85,B 0,C 180,E1 -18785.762,E2 -18785.762} C_VEL
LIN {X 0,Y 254.216,Z 586.444,A -85,B 0,C 180,E1 -18788.086,E2 -18788.086} C_VEL
LIN {X 0,Y 252.054,Z 595.392,A -85,B 0,C 180,E1 -18790.452,E2 -18790.452} C_VEL
LIN {X 0,Y 250.355,Z 603.389,A -85,B 0,C 180,E1 -18793.061,E2 -18793.061} C_VEL
LIN {X 0,Y 248.718,Z 610.869,A -85,B 0,C 180,E1 -18796.103,E2 -18796.103} C_VEL
LIN {X 0,Y 247.772,Z 615.612,A -85,B 0,C 180,E1 -18798.548,E2 -18798.548} C_VEL
LIN {X 0,Y 247.165,Z 620.529,A -85,B 0,C 180,E1 -18801.826,E2 -18801.826} C_VEL
LIN {X 0,Y 246.921,Z 623.931,A -85,B 0,C 180,E1 -18805.102,E2 -18805.102} C_VEL
LIN {X 0,Y 246.931,Z 625.919,A -85,B 0,C 180,E1 -18808.369,E2 -18808.369} C_VEL
LIN {X 0,Y 246.983,Z 626.398,A -85,B 0,C 180,E1 -18810,E2 -18810} C_VEL
LIN {X 0,Y 246.85,Z 626.337,A -85,B 0,C 180,E1 -18813.264,E2 -18813.264} C_VEL
LIN {X 0,Y 246.97,Z 624.942,A -85,B 0,C 180,E1 -18816.536,E2 -18816.536} C_VEL
LIN {X 0,Y 247.504,Z 622.192,A -85,B 0,C 180,E1 -18819.81,E2 -18819.81} C_VEL
LIN {X 0,Y 248.494,Z 618.014,A -85,B 0,C 180,E1 -18823.077,E2 -18823.077} C_VEL
LIN {X 0,Y 250.294,Z 612.294,A -85,B 0,C 180,E1 -18826.307,E2 -18826.307} C_VEL
LIN {X 0,Y 252.284,Z 605.966,A -85,B 0,C 180,E1 -18829.064,E2 -18829.064} C_VEL
LIN {X 0,Y 254.995,Z 597.9,A -85,B 0,C 180,E1 -18831.844,E2 -18831.844} C_VEL
LIN {X 0,Y 257.725,Z 589.587,A -85,B 0,C 180,E1 -18834.145,E2 -18834.145} C_VEL
LIN {X 0,Y 260.99,Z 579.594,A -85,B 0,C 180,E1 -18836.38,E2 -18836.38} C_VEL
LIN {X 0,Y 264.252,Z 568.485,A -85,B 0,C 180,E1 -18838.386,E2 -18838.386} C_VEL
LIN {X 0,Y 267.031,Z 557.457,A -85,B 0,C 180,E1 -18840.004,E2 -18840.004} C_VEL
LIN {X 0,Y 269.783,Z 545.499,A -85,B 0,C 180,E1 -18841.4,E2 -18841.4} C_VEL
LIN {X 0,Y 272.434,Z 532.293,A -85,B 0,C 180,E1 -18842.583,E2 -18842.583} C_VEL
LIN {X 0,Y 274.621,Z 518.612,A -85,B 0,C 180,E1 -18843.492,E2 -18843.492} C_VEL
LIN {X 0,Y 276.162,Z 504.817,A -85,B 0,C 180,E1 -18844.141,E2 -18844.141} C_VEL
LIN {X 0,Y 277.176,Z 487.366,A -85,B 0,C 180,E1 -18844.655,E2 -18844.655} C_VEL
LIN {X 0,Y 280.044,Z 421.421,A -85,B 0,C 180,E1 -18846.303,E2 -18846.303} C_VEL
LIN {X 0,Y 278.603,Z 413.363,A -85,B 0,C 180,E1 -18846.798,E2 -18846.798} C_VEL
LIN {X 0,Y 272.116,Z 398.763,A -85,B 0,C 180,E1 -18848.399,E2 -18848.399} C_VEL
LIN {X 0,Y 265.103,Z 384.914,A -85,B 0,C 180,E1 -18850.197,E2 -18850.197} C_VEL
LIN {X 0,Y 257.962,Z 372.137,A -85,B 0,C 180,E1 -18852.138,E2 -18852.138} C_VEL
LIN {X 0,Y 253.663,Z 365.471,A -85,B 0,C 180,E1 -18853.353,E2 -18853.353} C_VEL
LIN {X 0,Y 251.713,Z 361.832,A -85,B 0,C 180,E1 -18853.994,E2 -18853.994} C_VEL
LIN {X 0,Y 249.02,Z 353.085,A -85,B 0,C 180,E1 -18858.454,E2 -18858.454} C_VEL
LIN {X 0,Y 249.057,Z 353.086,A -85,B 0,C 180,E1 -18862.197,E2 -18862.197} C_VEL
LIN {X 0,Y 249.062,Z 353.085,A -85,B 0,C 180,E1 -18865.643,E2 -18865.643} C_VEL
LIN {X 0,Y 249.004,Z 353.088,A -85,B 0,C 180,E1 -18869.467,E2 -18869.467} C_VEL
LIN {X 0,Y 249.039,Z 353.081,A -85,B 0,C 180,E1 -18873.159,E2 -18873.159} C_VEL
LIN {X 0,Y 249.059,Z 353.082,A -85,B 0,C 180,E1 -18876.731,E2 -18876.731} C_VEL
LIN {X 0,Y 249.112,Z 353.08,A -85,B 0,C 180,E1 -18880.212,E2 -18880.212} C_VEL
LIN {X 0,Y 249.244,Z 353.059,A -85,B 0,C 180,E1 -18883.622,E2 -18883.622} C_VEL
LIN {X 0,Y 249.247,Z 353.061,A -85,B 0,C 180,E1 -18888.617,E2 -18888.617} C_VEL
LIN {X 0,Y 249.421,Z 353.027,A -85,B 0,C 180,E1 -18891.901,E2 -18891.901} C_VEL
LIN {X 0,Y 249.268,Z 353.056,A -85,B 0,C 180,E1 -18895.148,E2 -18895.148} C_VEL
LIN {X 0,Y 249.664,Z 353.007,A -85,B 0,C 180,E1 -18898.387,E2 -18898.387} C_VEL
LIN {X 0,Y 249.669,Z 352.996,A -85,B 0,C 180,E1 -18901.614,E2 -18901.614} C_VEL
LIN {X 0,Y 249.426,Z 353.025,A -85,B 0,C 180,E1 -18906.541,E2 -18906.541} C_VEL
LIN {X 0,Y 249.345,Z 353.05,A -85,B 0,C 180,E1 -18909.737,E2 -18909.737} C_VEL
LIN {X 0,Y 249.153,Z 353.074,A -85,B 0,C 180,E1 -18914.707,E2 -18914.707} C_VEL
LIN {X 0,Y 249.081,Z 353.082,A -85,B 0,C 180,E1 -18918.082,E2 -18918.082} C_VEL
LIN {X 0,Y 249.045,Z 353.078,A -85,B 0,C 180,E1 -18921.523,E2 -18921.523} C_VEL
LIN {X 0,Y 249.041,Z 353.079,A -85,B 0,C 180,E1 -18925.437,E2 -18925.437} C_VEL
LIN {X 0,Y 249.026,Z 353.061,A -85,B 0,C 180,E1 -18928.968,E2 -18928.968} C_VEL
LIN {X 0,Y 249.028,Z 353.073,A -85,B 0,C 180,E1 -18932.427,E2 -18932.427} C_VEL
LIN {X 0,Y 249.025,Z 353.062,A -85,B 0,C 180,E1 -18936.347,E2 -18936.347} C_VEL
LIN {X 0,Y 249.002,Z 353.182,A -85,B 0,C 180,E1 -18940.48,E2 -18940.48} C_VEL
LIN {X 0,Y 249.952,Z 355.886,A -85,B 0,C 180,E1 -18940.824,E2 -18940.824} C_VEL
LIN {X 0,Y 252.423,Z 358.726,A -85,B 0,C 180,E1 -18941.529,E2 -18941.529} C_VEL
LIN {X 0,Y 254.587,Z 361.985,A -85,B 0,C 180,E1 -18942.159,E2 -18942.159} C_VEL
LIN {X 0,Y 261.102,Z 371.548,A -85,B 0,C 180,E1 -18943.944,E2 -18943.944} C_VEL
LIN {X 0,Y 269.364,Z 385.918,A -85,B 0,C 180,E1 -18946.093,E2 -18946.093} C_VEL
LIN {X 0,Y 277.16,Z 401.553,A -85,B 0,C 180,E1 -18948.013,E2 -18948.013} C_VEL
LIN {X 0,Y 280.599,Z 409.648,A -85,B 0,C 180,E1 -18948.848,E2 -18948.848} C_VEL
LIN {X 0,Y 277.045,Z 487.756,A -85,B 0,C 180,E1 -18950.815,E2 -18950.815} C_VEL
LIN {X 0,Y 275.803,Z 501.879,A -85,B 0,C 180,E1 -18951.427,E2 -18951.427} C_VEL
LIN {X 0,Y 273.978,Z 515.252,A -85,B 0,C 180,E1 -18952.257,E2 -18952.257} C_VEL
LIN {X 0,Y 271.595,Z 528.297,A -85,B 0,C 180,E1 -18953.34,E2 -18953.34} C_VEL
LIN {X 0,Y 269.093,Z 540.743,A -85,B 0,C 180,E1 -18954.717,E2 -18954.717} C_VEL
LIN {X 0,Y 266.082,Z 552.443,A -85,B 0,C 180,E1 -18956.312,E2 -18956.312} C_VEL
LIN {X 0,Y 263.071,Z 563.224,A -85,B 0,C 180,E1 -18958.155,E2 -18958.155} C_VEL
LIN {X 0,Y 260.369,Z 572.672,A -85,B 0,C 180,E1 -18960.16,E2 -18960.16} C_VEL
LIN {X 0,Y 257.51,Z 581.274,A -85,B 0,C 180,E1 -18962.356,E2 -18962.356} C_VEL
LIN {X 0,Y 254.539,Z 589.892,A -85,B 0,C 180,E1 -18965.098,E2 -18965.098} C_VEL
LIN {X 0,Y 252.165,Z 596.815,A -85,B 0,C 180,E1 -18967.898,E2 -18967.898} C_VEL
LIN {X 0,Y 250.474,Z 601.583,A -85,B 0,C 180,E1 -18970.324,E2 -18970.324} C_VEL
LIN {X 0,Y 248.824,Z 606.496,A -85,B 0,C 180,E1 -18973.593,E2 -18973.593} C_VEL
LIN {X 0,Y 247.65,Z 609.897,A -85,B 0,C 180,E1 -18976.878,E2 -18976.878} C_VEL
LIN {X 0,Y 247.043,Z 611.894,A -85,B 0,C 180,E1 -18980.172,E2 -18980.172} C_VEL
LIN {X 0,Y 246.941,Z 612.542,A -85,B 0,C 180,E1 -18983.463,E2 -18983.463} C_VEL
LIN {X 0,Y 246.903,Z 611.87,A -85,B 0,C 180,E1 -18986.736,E2 -18986.736} C_VEL
LIN {X 0,Y 247.054,Z 609.872,A -85,B 0,C 180,E1 -18990,E2 -18990} C_VEL
LIN {X 0,Y 247.496,Z 606.508,A -85,B 0,C 180,E1 -18993.256,E2 -18993.256} C_VEL
LIN {X 0,Y 248.53,Z 601.669,A -85,B 0,C 180,E1 -18996.495,E2 -18996.495} C_VEL
LIN {X 0,Y 249.674,Z 597.002,A -85,B 0,C 180,E1 -18998.906,E2 -18998.906} C_VEL
LIN {X 0,Y 251.281,Z 590.007,A -85,B 0,C 180,E1 -19001.786,E2 -19001.786} C_VEL
LIN {X 0,Y 253.067,Z 581.867,A -85,B 0,C 180,E1 -19004.474,E2 -19004.474} C_VEL
LIN {X 0,Y 255.407,Z 573.103,A -85,B 0,C 180,E1 -19006.794,E2 -19006.794} C_VEL
LIN {X 0,Y 257.898,Z 562.506,A -85,B 0,C 180,E1 -19009.088,E2 -19009.088} C_VEL
LIN {X 0,Y 259.964,Z 552.96,A -85,B 0,C 180,E1 -19010.783,E2 -19010.783} C_VEL
LIN {X 0,Y 262.247,Z 541.497,A -85,B 0,C 180,E1 -19012.451,E2 -19012.451} C_VEL
LIN {X 0,Y 264.434,Z 528.918,A -85,B 0,C 180,E1 -19013.911,E2 -19013.911} C_VEL
LIN {X 0,Y 266.276,Z 515.925,A -85,B 0,C 180,E1 -19015.084,E2 -19015.084} C_VEL
LIN {X 0,Y 267.907,Z 501.883,A -85,B 0,C 180,E1 -19016.014,E2 -19016.014} C_VEL
LIN {X 0,Y 268.882,Z 488.041,A -85,B 0,C 180,E1 -19016.652,E2 -19016.652} C_VEL
LIN {X 0,Y 272.285,Z 401.171,A -85,B 0,C 180,E1 -19018.9,E2 -19018.9} C_VEL
LIN {X 0,Y 265.497,Z 384.666,A -85,B 0,C 180,E1 -19020.338,E2 -19020.338} C_VEL
LIN {X 0,Y 258.623,Z 370.201,A -85,B 0,C 180,E1 -19021.822,E2 -19021.822} C_VEL
LIN {X 0,Y 252.897,Z 360.401,A -85,B 0,C 180,E1 -19023.065,E2 -19023.065} C_VEL
LIN {X 0,Y 250.727,Z 356.891,A -85,B 0,C 180,E1 -19023.548,E2 -19023.548} C_VEL
LIN {X 0,Y 249.32,Z 354.376,A -85,B 0,C 180,E1 -19023.876,E2 -19023.876} C_VEL
LIN {X 0,Y 249.048,Z 353.087,A -85,B 0,C 180,E1 -19023.995,E2 -19023.995} C_VEL
LIN {X 0,Y 249.025,Z 353.09,A -85,B 0,C 180,E1 -19028.381,E2 -19028.381} C_VEL
LIN {X 0,Y 248.972,Z 353.095,A -85,B 0,C 180,E1 -19032.782,E2 -19032.782} C_VEL
LIN {X 0,Y 248.982,Z 353.094,A -85,B 0,C 180,E1 -19037.355,E2 -19037.355} C_VEL
LIN {X 0,Y 249.007,Z 353.09,A -85,B 0,C 180,E1 -19041.615,E2 -19041.615} C_VEL
LIN {X 0,Y 249.045,Z 353.087,A -85,B 0,C 180,E1 -19045.639,E2 -19045.639} C_VEL
LIN {X 0,Y 248.996,Z 353.093,A -85,B 0,C 180,E1 -19049.465,E2 -19049.465} C_VEL
LIN {X 0,Y 249.017,Z 353.08,A -85,B 0,C 180,E1 -19053.155,E2 -19053.155} C_VEL
LIN {X 0,Y 249.014,Z 353.085,A -85,B 0,C 180,E1 -19056.725,E2 -19056.725} C_VEL
LIN {X 0,Y 249.046,Z 353.052,A -85,B 0,C 180,E1 -19060.206,E2 -19060.206} C_VEL
LIN {X 0,Y 249.16,Z 353.072,A -85,B 0,C 180,E1 -19063.616,E2 -19063.616} C_VEL
LIN {X 0,Y 249.225,Z 353.025,A -85,B 0,C 180,E1 -19068.615,E2 -19068.615} C_VEL
LIN {X 0,Y 249.434,Z 353.028,A -85,B 0,C 180,E1 -19071.901,E2 -19071.901} C_VEL
LIN {X 0,Y 249.379,Z 353.042,A -85,B 0,C 180,E1 -19073.901,E2 -19073.901} C_VEL
LIN {X 0,Y 248.626,Z 353.137,A -85,B 0,C 180,E1 -19075.251,E2 -19075.251} C_VEL
LIN {X 0,Y 245.874,Z 353.479,A -85,B 0,C 180,E1 -19077.46,E2 -19077.46} C_VEL
LIN {X 0,Y 243.62,Z 353.763,A -85,B 0,C 180,E1 -19079.257,E2 -19079.257} C_VEL
LIN {X 0,Y 242.676,Z 353.872,A -85,B 0,C 180,E1 -19080.646,E2 -19080.646} C_VEL
LIN {X 0,Y 242.606,Z 353.88,A -85,B 0,C 180,E1 -19081.115,E2 -19081.115} C_VEL
LIN {X 0,Y 242.404,Z 353.912,A -85,B 0,C 180,E1 -19086.659,E2 -19086.659} C_VEL
LIN {X 0,Y 242.269,Z 353.925,A -85,B 0,C 180,E1 -19090.023,E2 -19090.023} C_VEL
LIN {X 0,Y 242.169,Z 353.94,A -85,B 0,C 180,E1 -19095.14,E2 -19095.14} C_VEL
LIN {X 0,Y 242.075,Z 353.95,A -85,B 0,C 180,E1 -19098.624,E2 -19098.624} C_VEL
LIN {X 0,Y 242.008,Z 353.959,A -85,B 0,C 180,E1 -19102.18,E2 -19102.18} C_VEL
LIN {X 0,Y 242.068,Z 353.953,A -85,B 0,C 180,E1 -19105.838,E2 -19105.838} C_VEL
LIN {X 0,Y 241.976,Z 353.966,A -85,B 0,C 180,E1 -19109.587,E2 -19109.587} C_VEL
LIN {X 0,Y 241.991,Z 353.968,A -85,B 0,C 180,E1 -19113.491,E2 -19113.491} C_VEL
LIN {X 0,Y 242.004,Z 353.968,A -85,B 0,C 180,E1 -19117.579,E2 -19117.579} C_VEL
LIN {X 0,Y 241.943,Z 353.976,A -85,B 0,C 180,E1 -19121.921,E2 -19121.921} C_VEL
LIN {X 0,Y 241.964,Z 354.092,A -85,B 0,C 180,E1 -19126.563,E2 -19126.563} C_VEL
LIN {X 0,Y 244.373,Z 362.53,A -85,B 0,C 180,E1 -19130.185,E2 -19130.185} C_VEL
LIN {X 0,Y 253.338,Z 380.282,A -85,B 0,C 180,E1 -19132.326,E2 -19132.326} C_VEL
LIN {X 0,Y 261.459,Z 398.893,A -85,B 0,C 180,E1 -19134.178,E2 -19134.178} C_VEL
LIN {X 0,Y 263.724,Z 405.086,A -85,B 0,C 180,E1 -19134.699,E2 -19134.699} C_VEL
LIN {X 0,Y 265.664,Z 420.779,A -85,B 0,C 180,E1 -19135.462,E2 -19135.462} C_VEL
LIN {X 0,Y 262.459,Z 500.594,A -85,B 0,C 180,E1 -19137.568,E2 -19137.568} C_VEL
LIN {X 0,Y 261.242,Z 514.568,A -85,B 0,C 180,E1 -19138.189,E2 -19138.189} C_VEL
LIN {X 0,Y 259.764,Z 526.541,A -85,B 0,C 180,E1 -19138.953,E2 -19138.953} C_VEL
LIN {X 0,Y 257.582,Z 540.274,A -85,B 0,C 180,E1 -19140.136,E2 -19140.136} C_VEL
LIN {X 0,Y 255.09,Z 553.366,A -85,B 0,C 180,E1 -19141.624,E2 -19141.624} C_VEL
LIN {X 0,Y 252.785,Z 564.59,A -85,B 0,C 180,E1 -19143.242,E2 -19143.242} C_VEL
LIN {X 0,Y 250.282,Z 575.099,A -85,B 0,C 180,E1 -19145.089,E2 -19145.089} C_VEL
LIN {X 0,Y 247.579,Z 585.991,A -85,B 0,C 180,E1 -19147.466,E2 -19147.466} C_VEL
LIN {X 0,Y 245.313,Z 594.981,A -85,B 0,C 180,E1 -19149.892,E2 -19149.892} C_VEL
LIN {X 0,Y 243.514,Z 602.713,A -85,B 0,C 180,E1 -19152.455,E2 -19152.455} C_VEL
LIN {X 0,Y 242.164,Z 608.696,A -85,B 0,C 180,E1 -19154.859,E2 -19154.859} C_VEL
LIN {X 0,Y 241.046,Z 613.846,A -85,B 0,C 180,E1 -19157.369,E2 -19157.369} C_VEL
LIN {X 0,Y 240.212,Z 619.167,A -85,B 0,C 180,E1 -19160.74,E2 -19160.74} C_VEL
LIN {X 0,Y 239.894,Z 622.14,A -85,B 0,C 180,E1 -19163.27,E2 -19163.27} C_VEL
LIN {X 0,Y 239.835,Z 623.781,A -85,B 0,C 180,E1 -19165.08,E2 -19165.08} C_VEL
LIN {X 0,Y 239.841,Z 625.69,A -85,B 0,C 180,E1 -19168.321,E2 -19168.321} C_VEL
LIN {X 0,Y 239.913,Z 626.185,A -85,B 0,C 180,E1 -19170,E2 -19170} C_VEL
LIN {X 0,Y 239.757,Z 626.152,A -85,B 0,C 180,E1 -19173.361,E2 -19173.361} C_VEL
LIN {X 0,Y 239.892,Z 624.782,A -85,B 0,C 180,E1 -19176.73,E2 -19176.73} C_VEL
LIN {X 0,Y 240.465,Z 622.057,A -85,B 0,C 180,E1 -19180.1,E2 -19180.1} C_VEL
LIN {X 0,Y 241.552,Z 617.906,A -85,B 0,C 180,E1 -19183.46,E2 -19183.46} C_VEL
LIN {X 0,Y 242.956,Z 613.825,A -85,B 0,C 180,E1 -19185.951,E2 -19185.951} C_VEL
LIN {X 0,Y 245.168,Z 607.027,A -85,B 0,C 180,E1 -19189.161,E2 -19189.161} C_VEL
LIN {X 0,Y 247.945,Z 599.118,A -85,B 0,C 180,E1 -19192.06,E2 -19192.06} C_VEL
LIN {X 0,Y 251.229,Z 589.61,A -85,B 0,C 180,E1 -19194.811,E2 -19194.811} C_VEL
LIN {X 0,Y 254.646,Z 579.664,A -85,B 0,C 180,E1 -19197.09,E2 -19197.09} C_VEL
LIN {X 0,Y 258.017,Z 568.62,A -85,B 0,C 180,E1 -19199.137,E2 -19199.137} C_VEL
LIN {X 0,Y 260.925,Z 557.657,A -85,B 0,C 180,E1 -19200.782,E2 -19200.782} C_VEL
LIN {X 0,Y 263.756,Z 545.8,A -85,B 0,C 180,E1 -19202.203,E2 -19202.203} C_VEL
LIN {X 0,Y 266.498,Z 532.782,A -85,B 0,C 180,E1 -19203.402,E2 -19203.402} C_VEL
LIN {X 0,Y 268.841,Z 518.594,A -85,B 0,C 180,E1 -19204.368,E2 -19204.368} C_VEL
LIN {X 0,Y 270.498,Z 504.111,A -85,B 0,C 180,E1 -19205.055,E2 -19205.055} C_VEL
LIN {X 0,Y 271.63,Z 484.957,A -85,B 0,C 180,E1 -19205.609,E2 -19205.609} C_VEL
LIN {X 0,Y 274.451,Z 422.718,A -85,B 0,C 180,E1 -19207.188,E2 -19207.188} C_VEL
LIN {X 0,Y 273.418,Z 416.554,A -85,B 0,C 180,E1 -19207.57,E2 -19207.57} C_VEL
LIN {X 0,Y 266.461,Z 400.786,A -85,B 0,C 180,E1 -19209.371,E2 -19209.371} C_VEL
LIN {X 0,Y 258.751,Z 385.688,A -85,B 0,C 180,E1 -19211.458,E2 -19211.458} C_VEL
LIN {X 0,Y 252.903,Z 375.596,A -85,B 0,C 180,E1 -19213.126,E2 -19213.126} C_VEL
LIN {X 0,Y 247.352,Z 366.54,A -85,B 0,C 180,E1 -19214.811,E2 -19214.811} C_VEL
LIN {X 0,Y 244.473,Z 361.966,A -85,B 0,C 180,E1 -19215.733,E2 -19215.733} C_VEL
LIN {X 0,Y 244.04,Z 360.694,A -85,B 0,C 180,E1 -19216.278,E2 -19216.278} C_VEL
LIN {X 0,Y 241.963,Z 353.965,A -85,B 0,C 180,E1 -19220.007,E2 -19220.007} C_VEL
